			350:
				(*1.发送给上位机的数据*)
			//	WorkStation_TCP.PLC_SEND1.m_nMoveState	:=2;			//send[9]//0-准备过程中 1-准备完成 2-曝光中 3-本次扫描结束	
				(*1.给上位机发送的数*)
				IF Entity_IO.bXrayExp THEN
					WorkStation_TCP.PLC_SEND1.m_nExpStates	:=2;//
				END_IF;
				WorkStation_TCP.PLC_SEND1.m_nScanProType:=2;			//send[16]
				
				(*2.曝光结束，跳出*)
				IF DT_Xray.RadExp_Step=66 THEN
					Step_Air:=360;	
				END_IF
			
			360:
				(*1.运动变量复位*)
				Entity_IO.bXaryOne:=FALSE;
				Entity_IO.bXaryTwo:=FALSE;
				Axis_QJ.QJ_AxisCmd.bAbs:=FALSE;
				Axis_XZ.XZ_AxisCmd.bAbs:=FALSE;	
				Entity_IO.bTriggerOut:=FALSE;
	
				(*2.给上位机发送数据，不能太快*)
				TON_Air[36](IN:=TRUE , PT:=T#1600MS , Q=> , ET=> );	//留些时间给上位机发送本次扫描结束方案标志
				
				(*2.扫描结束，发送结束标志位*)
				IF DT_Xray.RadExp_Step=77 THEN 
					WorkStation_TCP.PLC_SEND1.m_nMoveState:=3;			//send[9] //0-准备过程中 1-准备完成 2-曝光中 3-本次扫描结束
				END_IF;
				
				(*3.判断师傅最后一次扫描*)
				IF TON_Air[36].Q THEN
					IF (WorkStation_TCP.PLC_RECV1.m_nCircleIndex+1)>=(WorkStation_TCP.PLC_RECV1.m_nCircleCount) AND bAirLast3 AND DT_Xray.RadExp_Step=77 THEN 	//用于区分自动扫是否最后一次，此时=1，=1都等于1
						GVL_SCAN.bJumpScan:=TRUE;
					END_IF;
				END_IF
				
				(*4.不是最后一次，收到下一次命令，继续扫*)
				IF WorkStation_TCP.PLC_RECV1.m_nSocketType=1 AND DT_Xray.RadExp_Step=77 THEN 	//增加第二次运动判断，m_nSocketType=1 
					Step_Air:=300;
				END_IF
	END_CASE
END_ACTION

TRANSITION T_AirCal:
(*进入空气校正/高清校正模式*)
	WorkStation_TCP.PLC_RECV1.m_nSocketType=1 AND (WorkStation_TCP.PLC_RECV1.m_nExpId=7  OR WorkStation_TCP.PLC_RECV1.m_nExpId=8)
END_TRANSITION

TRANSITION T_AirCal_Quick:
(*进入空气校正/快速校正模式*)
	WorkStation_TCP.PLC_RECV1.m_nSocketType=1 AND WorkStation_TCP.PLC_RECV1.m_nExpId=8
END_TRANSITION

ACTION _AirCalQuick_active:

	CASE Step_Air_Quick OF 
		300://快速扫描校正
				//初始化准备流程
				(*1.给上位机发送的数据*)
				WorkStation_TCP.PLC_SEND1.m_nMoveState:=0;			//send[9] //0-准备过程中 1-准备完成 2-曝光中 3-本次扫描结束 
				bAirLast3		:=FALSE;
				Entity_IO.bXraySwitch:=FALSE;//
				(*2.中间变量复位*)
				FOR i:=1 TO 50 BY 1 DO 
					TON_Air[i](IN:= FALSE);
				END_FOR
				Axis_XZ.XZ_AxisCmd.bAbs		:=FALSE;
				Axis_QJ.QJ_AxisCmd.bAbs		:=FALSE;
				Step_Air_Quick:=310;
				
			310:
				(*1.发送给上位机的数据*)
				WorkStation_TCP.PLC_SEND1.m_nExpStates	:=1;		//0-准备过程中 1-准备完成 2-曝光中 3-本次扫描结束	
				WorkStation_TCP.PLC_SEND1.m_nMoveState	:=0;		//起始、终止状态， 默认值0， 1为当前扫描方案处于准备好状态，可以准备扫描；2为当前扫描方案结束，运动过程中值为0
				WorkStation_TCP.PLC_SEND1.m_nScanProType:=2;		//扫描方案类型 , 1-手动，0-自动. 
			
				(*2.旋转轴和前进轴自动运动到目标位置*)
				(*2.1 旋转轴直接运动到目标位置*)
				Axis_XZ.XZ_AxisCmd.AxisPara.rAbsPosition	:=LIMIT(-3,WorkStation_TCP.PLC_RECV1.m_nRotateBegin,363);
				Axis_XZ.XZ_AxisCmd.AxisPara.rAbsVelocity	:=30;
				TON_Air[31](IN:=TRUE , PT:=T#500MS);
				Axis_XZ.XZ_AxisCmd.bAbs						:=TON_Air[31].Q;
	
				(*2.2 前进轴直接运动到目标位置*)
				Axis_QJ.QJ_AxisCmd.AxisPara.rAbsPosition	:=LIMIT(0,WorkStation_TCP.PLC_RECV1.m_fScanTop,900);
				Axis_QJ.QJ_AxisCmd.AxisPara.rAbsVelocity	:=60;
				TON_Air[32](IN:=TRUE , PT:=T#500MS);
				Axis_QJ.QJ_AxisCmd.bAbs						:=TON_Air[32].Q;
				
				(*5.跳转*)
				TON_Air[33](IN:=ABS(Axis_QJ.QJ_AxisState.rActPosition-WorkStation_TCP.PLC_RECV1.m_fScanTop)<1 
					AND ABS(Axis_XZ.XZ_AxisState.rActPosition-WorkStation_TCP.PLC_RECV1.m_nRotateBegin)<1 
					AND Axis_XZ.XZ_AxisState.bStandStill AND Axis_QJ.QJ_AxisState.bStandStill, PT:=T#150MS);
				IF TON_Air[33].Q THEN  
					Step_Air_Quick:=320;
				END_IF
				
			320://写入射线源参数成功
				(*1.变量复位*)
				Axis_XZ.XZ_AxisCmd.bAbs		:=FALSE;
				Axis_QJ.QJ_AxisCmd.bAbs		:=FALSE;
				
				(*2.射线源参数写入正常完毕*)
				IF DT_Xray.ExpPara_Step=66 THEN
					Step_Air_Quick:=330;
				END_IF
				
			330:
				//扫描中间态，跳转使用
				(*1.变量复位*)
				FOR i:=1 TO 50 BY 1 DO 
					TON_Air[i](IN:= FALSE);
				END_FOR
				Axis_QJ.QJ_AxisCmd.bAbs:=FALSE;//复位前进轴
				Axis_XZ.XZ_AxisCmd.bAbs:=FALSE;//复位旋转轴
				Step_Air_Quick:=340;
				
			340://开启曝光
				(*1.发送给上位机的数据*)
				WorkStation_TCP.PLC_SEND1.m_nMoveState	:=1;	//send[9]
				WorkStation_TCP.PLC_SEND1.m_nScanProType:=2;	//send[16]
				
				(*2.射线源参数写入成功，开启透视*)
				IF DT_Xray.ExpPara_Step=66 THEN  //保证写入参数
					Entity_IO.bXaryOne:=TRUE;//开启一二档
					Entity_IO.bXaryTwo:=TRUE;//开启一二档
				END_IF;
				
				(*3.判断是否最后一次扫描*)
				IF WorkStation_TCP.PLC_RECV1.m_nLastMsg=1 THEN
					bAirLast3 := TRUE;
				ELSE
					bAirLast3 := FALSE;
				END_IF
				
				(*4.跳转指令*)
				TON_Air[34](IN:=TRUE,PT:=T#2600MS);//把曝光的时间加这这里了
				IF TON_Air[34].Q AND Entity_IO.bXaryOne AND Entity_IO.bXaryTwo THEN
					Step_Air_Quick:=350;
				END_IF
				
			350:
				(*1.发送给上位机的数据*)
				WorkStation_TCP.PLC_SEND1.m_nMoveState	:=2;			//send[9]//0-准备过程中 1-准备完成 2-曝光中 3-本次扫描结束	
				WorkStation_TCP.PLC_SEND1.m_nScanProType:=2;			//send[16]
				
				(*2.曝光结束，跳出*)
				IF DT_Xray.RadExp_Step=66 THEN
					Step_Air_Quick:=360;	
				END_IF
			
			360:
				(*1.运动变量复位*)
				Entity_IO.bXaryOne:=FALSE;
				Entity_IO.bXaryTwo:=FALSE;
				Axis_QJ.QJ_AxisCmd.bAbs:=FALSE;
				Axis_XZ.XZ_AxisCmd.bAbs:=FALSE;	
				Entity_IO.bTriggerOut:=FALSE;
	
				(*2.给上位机发送数据，不能太快*)
				TON_Air[36](IN:=TRUE , PT:=T#1600MS , Q=> , ET=> );	//留些时间给上位机发送本次扫描结束方案标志
				
				(*2.扫描结束，发送结束标志位*)
				IF DT_Xray.RadExp_Step=77 THEN 
					WorkStation_TCP.PLC_SEND1.m_nMoveState:=3;			//send[9] //0-准备过程中 1-准备完成 2-曝光中 3-本次扫描结束
				END_IF;
				
				(*3.判断师傅最后一次扫描*)
				IF TON_Air[36].Q THEN
					IF (WorkStation_TCP.PLC_RECV1.m_nCircleIndex+1)>=(WorkStation_TCP.PLC_RECV1.m_nCircleCount) AND bAirLast3 AND DT_Xray.RadExp_Step=77 THEN 	//用于区分自动扫是否最后一次，此时=1，=1都等于1
						GVL_SCAN.bJumpScan:=TRUE;
					END_IF;
				END_IF
				
				(*4.不是最后一次，收到下一次命令，继续扫*)
				IF WorkStation_TCP.PLC_RECV1.m_nSocketType=1 AND DT_Xray.RadExp_Step=77 THEN 	//增加第二次运动判断，m_nSocketType=1 
					Step_Air_Quick:=300;
				END_IF
		END_CASE
END_ACTION

ACTION _AirCalQuick_entry:
Step_Air_Quick:=300; 

GVL_State.iPLC_State:=350;//空气校正
END_ACTION

ACTION _AirCalHign_exit:


	Entity_IO.bTriggerOut:=FALSE;
	Entity_io.bXraySwitch:=FALSE;//PF CLK信号切换继电器 不得电是默认BUCKY触发
	
	iTriggerNum1:=0;
	iTriggerNum2:=0;
END_ACTION

ACTION _AirCalQuick_exit:

END_ACTION

ACTION _a_Debug_exit:


Entity_IO.bXaryFlu:=FALSE;
END_ACTION

ACTION _a_Emergercy_exit:

Axis_XZ.XZ_AxisCmd.bReset:=TRUE;
Axis_QJ.QJ_AxisCmd.bReset:=TRUE;
END_ACTION

ACTION _ModeWait_active:

IF Axis_XZ.XZ_AxisCmd.bPower=FALSE THEN 
	Axis_XZ.XZ_AxisCmd.bPower:=TRUE;
ELSE
	;
END_IF

IF Axis_QJ.QJ_AxisCmd.bPower=FALSE THEN 
	Axis_QJ.QJ_AxisCmd.bPower:=TRUE;
ELSE
	;
END_IF
END_ACTION

END_PROGRAM

// Device/Application/Refer/XRAY_RS485
PROGRAM XRAY_RS485
VAR
	Open_0: COM.Open;Hulala:BOOL;
	Write_0: COM.Write;
	Read_0: COM.Read;
	Close_0: COM.Close;
	xOpen_Exe:BOOL;
	hComHandle:CAA.HANDLE;
	byWrite2:ARRAY [0..3] OF BYTE;
	byWrite3:ARRAY [0..4] OF BYTE;
	byWrite4:ARRAY [0..5] OF BYTE;
	byWrite5:ARRAY [0..6] OF BYTE;
	byWrite6:ARRAY [0..7] OF BYTE;
	byWrite7:ARRAY [0..8] OF BYTE;
	byWrite8:ARRAY [0..9] OF BYTE;
	byWrite9:ARRAY [0..10] OF BYTE;
	xWrite_Exe:BOOL;
	xRead_Exe:BOOL;
    byReadData:ARRAY [0..255] OF BYTE;
    xClose_Exe:BOOL;
	aParamsB19200 : ARRAY [1..7] OF COM.PARAMETER := [
    (udiParameterId := COM.CAA_Parameter_Constants.udiPort,udiValue := 3), 					//指令端口2,3,4,5分别对应硬件接口com2、com0、com1、com3
    (udiParameterId := COM.CAA_Parameter_Constants.udiBaudrate,udiValue := 19200),			//波特率，设置为19200
    (udiParameterId := COM.CAA_Parameter_Constants.udiParity,udiValue := COM.PARITY.NONE),	//校验，设置为无校验
    (udiParameterId := COM.CAA_Parameter_Constants.udiStopBits,udiValue := COM.STOPBIT.ONESTOPBIT),//停止位，1位
    (udiParameterId := COM.CAA_Parameter_Constants.udiTimeout,udiValue := 500),				//超时时间，设置成500ms
    (udiParameterId := COM.CAA_Parameter_Constants.udiByteSize,udiValue := 8),				//数据位
    (udiParameterId := COM.CAA_Parameter_Constants.udiBinary, udiValue := 1)				//二进制参数，启用二进制模式
];		
	TON1,TON2:Standard.TON;
	bSend:BOOL;
	iSize	:INT;
	String2Byte1:String2Byte;
	sSendString:STRING;//
	BLINK1,BLINK2:Blink;
//	Main_Step,Init_Step,DefaultPara_Step,Standby_Step,Rad_Step,Lookup_Step:UINT;
	sRecvString:ARRAY [0..9] OF STRING;	
	sRecvByte:ARRAY [0..39] OF BYTE;	
	i:INT;
	RecvNum,RecvNum1:INT;
	ASCII_Chart_N1:ARRAY [0..9] OF ASCII_Chart_N;
	sRecvStringA1,sRecvStringA2,sRecvStringA3,sRecvStringA4:STRING;
	sRecvStringA5,sRecvStringA6,sRecvStringA7,sRecvStringA0:STRING;
	R_TRIG1:Standard.R_TRIG;
	R30_0,R30_1,R30_2,R30_3,R30_4,R30_5,R30_6:Standard.R_TRIG;
	R10,R20,R30,R40,R50,R60:Standard.R_TRIG;
	TON0_20,TON30_0,TON30_20,TON30_30:Standard.TON;
	f10:F_TRIG;
	BLINK1_ST,BLINK11: BLINK;
	TEMP_MA:UINT;
	TEMP_MS: UINT;
	TON3,TON_ST,TON40,TON_FLR:TON;
	ASCII_Chart_N2:ARRAY[0..30] OF ASCII_Chart_N;
	ASCII_Chart_N_Alarm:ARRAY[0..5] OF ASCII_Chart_N;
	TEMP_FLX1:BOOL;
	TON22:TON;
	R_JUMP20:R_TRIG;
	TON33: TON;
	TON_DelayPara:TON;
	HULALA111:BOOL;
	
	TON11,TON12:TON;
	TON_KV,TON_MA:Standard.TON; //参数设置不对后，延迟进行报警处理0228
	Booting: BOOL;
	hlaldjlk: BOOL;
	Feedback_mA1:REAL;
	Feedback_Kv1:UDINT;
	TON_DELAY:TON;
	
	XXX:X_RayFluPara;
	aaa1:ARRAY[1..255] OF BYTE;
	aaa:ARRAY[1..255] OF BYTE;
	
ddd:UINT;
Error:INT;
j:INT;
xxxxx:String_TO_ASCII;
	CheckSum:UINT;
	CheckSum1: UINT;
	CheckSum3:STRING;
	sSendStringX:STRING;
	
	
	ReadString:RecvStringS;
	
	
END_VAR

VAR_INPUT
	
END_VAR

VAR_OUTPUT
	Main_Step,Init_Step,DefaultPara_Step,Standby_Step,Rad_Step,Lookup_Step:UINT;
	Feedback_Kv:UDINT;
	Feedback_mA:REAL;
	Feedback_ms:REAL;
	Feedback_nFocus:UDINT;
	Feedback_nMHuValue:REAL;
	Feedback_AccTime:REAL;
	iAlarmNum:UINT;		//射线源部分的报警位
END_VAR

(*README*)
(*射线源通讯子功能块*)

(*---------------------------------------------------第一部分：串口参数设置------------------------------------------------*)
(*1.open*)
	TON1(IN:=TRUE , PT:=T#5S);//开机后5秒打开串口
	Open_0(xExecute:=TON1.Q , xDone=> , xBusy=> , xError=> , usiListLength:=20 , pParameterList:=ADR(aParamsB19200) , eError=> , hCom=>hComHandle );

	
(*2.Write*)
	Write_0(
			xExecute:= Open_0.xDone AND bSend, 
			xAbort:= , 
			udiTimeOut:=500 , 
			xDone=> , 
			xBusy=> , 
			xError=> , 
			xAborted=> , 
			hCom:= hComHandle, 
			pBuffer:= , //后面写的
			szSize:= , 
			eError=> );	
			
(*3.Read*)
	TON2(IN:=NOT TON2.Q , PT:=T#20MS , Q=> , ET=> );	//射线源周期100ms
	Read_0(
			xExecute:= Open_0.xDone AND TON2.Q AND NOT(bSend),
			xAbort:= , 
			udiTimeOut:= 500, 
			xDone=> , 
			xBusy=> , 
			xError=> , 
			xAborted=> , 
			hCom:= hComHandle, 
			pBuffer:= ADR(byReadData), 
			szBuffer:= 10, 
			eError=> , 
			szSize=> );
	
(*4.Close*)
	Close_0(
			xExecute:= xClose_Exe, 
			xDone=> , 
			xBusy=> , 
			xError=> , 
			hCom:= hComHandle, 
			eError=> );

(*--------------------------------------------第二部分，数据处理--------------------------------------------------*)
(*2.1 写入命令处理*)
	iSize:=LIMIT(0,LEN(sSendString),255); 		//获取写入的字符串长度	已增加03H结束符+CheckSum和校验	
	Write_0.szSize:=INT_TO_USINT(iSize);
	Write_0.pBuffer:=ADR(sSendString);

	XXX( 
	WS:= 1, 
	FLF:= 2, 
	FLA:=0 , 
	FLS:=195 , 
	FLR:=1 , 
	FLK:= 090, 
	FLM:= 060, 
	Out=> );
	
	sSendStringX:=XXX.Out;

xxxxx(
		InputString:=XXX.Out , 
		MaxArraySize:= 255, 
		ASCIIArray=> aaa1, 
		ArrayLength=> , 
		Error=> , 
		ErrorMessage=> );
		
	CheckSum:=0;
	FOR j:=1 TO 255 BY 1 DO
		IF aaa1[j]=16#20 THEN   	//空格对应的ASCII码不计入和校验中
			CONTINUE;
		END_IF
		CheckSum:=CheckSum+aaa1[j];
	END_FOR

	CheckSum1:=(CheckSum) AND 16#FF; 	//取低字节byte
	IF CheckSum1<16 THEN 
		NumToHexString(In:= CheckSum1, L:=1, Fill:=LS_OmronUtils._eFILL_CHR._ZERO, Out=> CheckSum3);
	ELSE
		NumToHexString(In:= CheckSum1, L:=2, Fill:=LS_OmronUtils._eFILL_CHR._NULL, Out=> CheckSum3);
	END_IF
	
	sSendString:=CONCAT(STR1:=sSendStringX , STR2:= CheckSum3);


	ReadString(Excute:= Read_0.xDone AND Read_0.szSize<>0, Size:=__UXINT_TO_INT(Read_0.szSize) , RecvArray:=byReadData , RecvString=>sRecvStringA0 );









(*

(*2.1 写入命令处理*)
	iSize:=LIMIT(0,LEN(sSendString),10); 		//获取写入的字符串长度	已增加03H结束符+CheckSum和校验	
	String2Byte1(sXrayString:=sSendString , sByte=> );
	Write_0.szSize:=INT_TO_USINT(iSize)+2;
	CASE iSize OF 
	2:
		(*2个字符的命令*)	
		byWrite2[0]:=String2Byte1.sByte[1];
		byWrite2[1]:=String2Byte1.sByte[2];
		byWrite2[2]:=16#03;
		byWrite2[3]:=byWrite2[0]+byWrite2[1]+byWrite2[2];
		Write_0.pBuffer:=ADR(byWrite2);
	3:	
		(*3个字符的命令*)	
		byWrite3[0]:=String2Byte1.sByte[1];
		byWrite3[1]:=String2Byte1.sByte[2];
		byWrite3[2]:=String2Byte1.sByte[3];
		byWrite3[3]:=16#03;
		byWrite3[4]:=byWrite3[0]+byWrite3[1]+byWrite3[2]+byWrite3[3];
		Write_0.pBuffer:=ADR(byWrite3);
	
	4:
		(*4个字符的命令*)	
		byWrite4[0]:=String2Byte1.sByte[1];
		byWrite4[1]:=String2Byte1.sByte[2];
		byWrite4[2]:=String2Byte1.sByte[3];
		byWrite4[3]:=String2Byte1.sByte[4];
		byWrite4[4]:=16#03;
		byWrite4[5]:=byWrite4[0]+byWrite4[1]+byWrite4[2]+byWrite4[3]+byWrite4[4];
		Write_0.pBuffer:=ADR(byWrite4);
	
	5:
		(*5个字符的命令*)	
		byWrite5[0]:=String2Byte1.sByte[1];
		byWrite5[1]:=String2Byte1.sByte[2];
		byWrite5[2]:=String2Byte1.sByte[3];
		byWrite5[3]:=String2Byte1.sByte[4];
		byWrite5[4]:=String2Byte1.sByte[5];
		byWrite5[5]:=16#03;
		byWrite5[6]:=byWrite5[0]+byWrite5[1]+byWrite5[2]+byWrite5[3]+byWrite5[4]+byWrite5[5];
		Write_0.pBuffer:=ADR(byWrite5);
		
	6:
		(*6个字符的命令*)	
		byWrite6[0]:=String2Byte1.sByte[1];
		byWrite6[1]:=String2Byte1.sByte[2];
		byWrite6[2]:=String2Byte1.sByte[3];
		byWrite6[3]:=String2Byte1.sByte[4];
		byWrite6[4]:=String2Byte1.sByte[5];
		byWrite6[5]:=String2Byte1.sByte[6];
		byWrite6[6]:=16#03;
		byWrite6[7]:=byWrite6[0]+byWrite6[1]+byWrite6[2]+byWrite6[3]+byWrite6[4]+byWrite6[5]+byWrite6[6];
		Write_0.pBuffer:=ADR(byWrite6);		
	7:
		(*7个字符的命令*)	
		byWrite7[0]:=String2Byte1.sByte[1];
		byWrite7[1]:=String2Byte1.sByte[2];
		byWrite7[2]:=String2Byte1.sByte[3];
		byWrite7[3]:=String2Byte1.sByte[4];
		byWrite7[4]:=String2Byte1.sByte[5];
		byWrite7[5]:=String2Byte1.sByte[6];
		byWrite7[6]:=String2Byte1.sByte[7];
		byWrite7[7]:=16#03;
		byWrite7[8]:=byWrite7[0]+byWrite7[1]+byWrite7[2]+byWrite7[3]+byWrite7[4]+byWrite7[5]+byWrite7[6]+byWrite7[7];
		Write_0.pBuffer:=ADR(byWrite7);
		
	8:(*8个字符的命令*)	
		byWrite8[0]:=String2Byte1.sByte[1];
		byWrite8[1]:=String2Byte1.sByte[2];
		byWrite8[2]:=String2Byte1.sByte[3];
		byWrite8[3]:=String2Byte1.sByte[4];
		byWrite8[4]:=String2Byte1.sByte[5];
		byWrite8[5]:=String2Byte1.sByte[6];
		byWrite8[6]:=String2Byte1.sByte[7];
		byWrite8[7]:=String2Byte1.sByte[8];
		byWrite8[8]:=16#03;
		byWrite8[9]:=byWrite8[0]+byWrite8[1]+byWrite8[2]+byWrite8[3]+byWrite8[4]+byWrite8[5]+byWrite8[6]+byWrite8[7]+byWrite8[8];
		Write_0.pBuffer:=ADR(byWrite8);
	ELSE
		;//输入错误
	END_CASE
	
*)		
	(*2.2 读取命令*)
(*	sRecvByte:=byReadData;

	R_TRIG1(CLK:=Read_0.xDone AND Read_0.szSize<>0, Q=> );		//获取读到了多少个字符
	IF R_TRIG1.Q THEN
		RecvNum:=LIMIT(0,__UXINT_TO_INT(Read_0.szSize)-2,9);	//限制了一下字符0124
	END_IF;

	FOR i:=0 TO RecvNum BY 1 DO 
		ASCII_Chart_N1[i](byASCII:=sRecvByte[i] , sOut_Single=>sRecvString[i] );//需要调用功能块才能有输出
	END_FOR 

	CASE RecvNum OF 		//最长8个字符,如遇到RS和RR的反馈，就自己数字节吧，这里给反馈命令使用
		0:
			sRecvStringA0:='NULL';
		1:
			sRecvStringA0:=sRecvString[0];
		2:
			sRecvStringA0:=CONCAT(STR1:=sRecvString[0] , STR2:= sRecvString[1]);
		3:
			sRecvStringA1:=CONCAT(STR1:=sRecvString[0] , STR2:= sRecvString[1]);
			sRecvStringA0:=CONCAT(STR1:=sRecvStringA1 , STR2:= sRecvString[2]);
		4:
			sRecvStringA1:=CONCAT(STR1:=sRecvString[0] , STR2:= sRecvString[1]);
			sRecvStringA2:=CONCAT(STR1:=sRecvString[2] , STR2:= sRecvString[3]);
			sRecvStringA0:=CONCAT(STR1:=sRecvStringA1 , STR2:= sRecvStringA2);
		5:
			sRecvStringA1:=CONCAT(STR1:=sRecvString[0] , STR2:= sRecvString[1]);
			sRecvStringA2:=CONCAT(STR1:=sRecvString[2] , STR2:= sRecvString[3]);
			sRecvStringA3:=CONCAT(STR1:=sRecvStringA1 , STR2:= sRecvStringA2);
			sRecvStringA0:=CONCAT(STR1:=sRecvStringA3 , STR2:= sRecvString[4]);
		6:
			sRecvStringA1:=CONCAT(STR1:=sRecvString[0] , STR2:= sRecvString[1]);
			sRecvStringA2:=CONCAT(STR1:=sRecvString[2] , STR2:= sRecvString[3]);
			sRecvStringA3:=CONCAT(STR1:=sRecvString[4] , STR2:= sRecvString[5]);
			sRecvStringA4:=CONCAT(STR1:=sRecvStringA1 , STR2:= sRecvStringA2);
			sRecvStringA0:=CONCAT(STR1:=sRecvStringA4 , STR2:= sRecvStringA3);
		7:
			sRecvStringA1:=CONCAT(STR1:=sRecvString[0] , STR2:= sRecvString[1]);
			sRecvStringA2:=CONCAT(STR1:=sRecvString[2] , STR2:= sRecvString[3]);
			sRecvStringA3:=CONCAT(STR1:=sRecvString[4] , STR2:= sRecvString[5]);
			sRecvStringA4:=CONCAT(STR1:=sRecvStringA1 , STR2:= sRecvStringA2);
			sRecvStringA5:=CONCAT(STR1:=sRecvStringA4 , STR2:= sRecvStringA3);
			sRecvStringA0:=CONCAT(STR1:=sRecvStringA5 , STR2:= sRecvString[6]);
		8:
			sRecvStringA1:=CONCAT(STR1:=sRecvString[0] , STR2:= sRecvString[1]);
			sRecvStringA2:=CONCAT(STR1:=sRecvString[2] , STR2:= sRecvString[3]);
			sRecvStringA3:=CONCAT(STR1:=sRecvString[4] , STR2:= sRecvString[5]);
			sRecvStringA4:=CONCAT(STR1:=sRecvString[6] , STR2:= sRecvString[7]);
			sRecvStringA5:=CONCAT(STR1:=sRecvStringA1 , STR2:= sRecvStringA2);
			sRecvStringA6:=CONCAT(STR1:=sRecvStringA3 , STR2:= sRecvStringA4);
			sRecvStringA0:=CONCAT(STR1:=sRecvStringA5 , STR2:= sRecvStringA6);
		9:
			sRecvStringA1:=CONCAT(STR1:=sRecvString[0] , STR2:= sRecvString[1]);
			sRecvStringA2:=CONCAT(STR1:=sRecvString[2] , STR2:= sRecvString[3]);
			sRecvStringA3:=CONCAT(STR1:=sRecvString[4] , STR2:= sRecvString[5]);
			sRecvStringA4:=CONCAT(STR1:=sRecvString[6] , STR2:= sRecvString[7]);
			sRecvStringA5:=CONCAT(STR1:=sRecvStringA1 , STR2:= sRecvStringA2);
			sRecvStringA6:=CONCAT(STR1:=sRecvStringA3 , STR2:= sRecvStringA4);
			sRecvStringA7:=CONCAT(STR1:=sRecvStringA5 , STR2:= sRecvStringA6);
			sRecvStringA0:=CONCAT(STR1:=sRecvStringA7 , STR2:= sRecvString[8]);
		ELSE
			sRecvStringA0:='Too Long';
	END_CASE
*)
(*3.射线源状态机处理*)	
//	AXray( );
//	GVL_State.iXray_State:=UINT_TO_BYTE(Main_Step);//获取射线源状态

ACTION AXray:

(*---------------------------------------------第三部分：射线源状态机---------------------------------------------------*)
(*0.公共部分*)
(*	BLINK1(ENABLE:=TON1.Q , TIMELOW:=T#300MS , TIMEHIGH:=T#200MS , OUT=> );
	BLINK1_ST(ENABLE:=TON1.Q , TIMELOW:=T#2S , TIMEHIGH:=T#2S , OUT=> );
	
	(*1.初始化阶段，Initialization Phase*)
			CASE Main_Step OF 
				0:	(*1.初始化阶段，Initialization Phase*)
				IF (sRecvByte[0]= 16#45 AND sRecvByte[1]= 16#4C) OR sRecvStringA0='ST008' THEN //收到ER或EL,确认收到了错误信号，ER可以理解为可恢复，EL为不可恢复 收到EL信号可复位，ER信号只是显示
						Main_Step:=40;
				ELSE
					CASE Init_Step OF 
					0:	//参数初始化
						bSend			:=FALSE;
						DefaultPara_Step:=0;
						Standby_Step	:=0;
						Rad_Step		:=0;//射线步骤复位
						TON11(IN:= TRUE, PT:=T#3S);//开机延迟
						IF TON11.Q THEN
							Init_Step		:=10;
						END_IF
						
					10:	//建立通讯
						TON11(IN:= FALSE);
						sSendString:='ST';
						bSend:=BLINK1_ST.OUT;  
						IF sRecvStringA0='ST001' OR sRecvStringA0='ST002' THEN //收到ST000，通讯正常//此版本是001，所有状态都加1，文档状态说明都加1
							Init_Step:=20;
						ELSE
							iAlarmNum:=301;		//通讯错误
						END_IF
						
					20://检查错误,如果有错误，就复位，没错误，延迟2秒跳转
						iAlarmNum:=0;		//通讯
						IF sRecvByte[0]= 16#45 AND (sRecvByte[1]= 16#4C) THEN //收到ER或EL,确认收到了错误信号，EL可以理解为可恢复，ER为不可恢复 收到EL信号可复位，ER信号只是显示
							sSendString:=sRecvStringA0;
							bSend:=BLINK1.OUT;
							TON0_20(IN:=FALSE);
						ELSE
							TON0_20(IN:=TRUE , PT:=T#2S);//2秒内无报错
							IF TON0_20.Q THEN
								sSendString:='ST';
								bSend:=BLINK1.OUT;
								IF sRecvStringA0='ST002' OR sRecvStringA0='ST001' THEN //收到ST002，通讯正常//此版本是001，所有状态都加1
									Init_Step:=66;
								END_IF
							END_IF;
						END_IF
					66:
						Main_Step:=10;
					ELSE
						;
					END_CASE
				END_IF;
				
				10:	(*写入默认参数，开机只写一次*)	
					IF (sRecvByte[0]= 16#45 AND sRecvByte[1]= 16#4C) OR sRecvStringA0='ST008' THEN //收到ER或EL,确认收到了错误信号，ER可以理解为可恢复，EL为不可恢复 收到EL信号可复位，ER信号只是显示
						Main_Step:=40;
					ELSE
						CASE DefaultPara_Step OF 
						0:
							bSend:=FALSE;
							TON_DelayPara(IN:=FALSE);
							DefaultPara_Step:=5;
					
						5:
							TON_DelayPara(IN:=TRUE , PT:=T#5S , Q=> , ET=> );//写默认参数的时候需要等等射线源一些时间
							IF TON_DelayPara.Q THEN
								DefaultPara_Step:=10;
							END_IF
							
						10://1.关闭AEC
							TON_DelayPara(IN:=FALSE);
							sSendString:='FI000';
							bSend:=BLINK1.OUT;
							IF sRecvStringA0='FI000' THEN
								DefaultPara_Step:=20;
							END_IF
							
						20:
							sSendString:='ET1';
							bSend:=BLINK1.OUT;
							IF sRecvStringA0='ET1' THEN
								DefaultPara_Step:=30;
							END_IF
							
						30://工作模式选择
							sSendString:='WS1';
							bSend:=BLINK1.OUT;
							IF sRecvStringA0='WS1' THEN
								DefaultPara_Step:=40;
							END_IF
						40:
							bSend:=FALSE;
							Main_Step:=20;
						ELSE 
							;
						END_CASE
					END_IF;
		
				20:	(*静止等待状态，Standby Phase*)//注意增加ST，每5秒的周期
					Rad_Step	:=0;
					IF (sRecvByte[0]= 16#45 AND sRecvByte[1]= 16#4C) OR sRecvStringA0='ST008' THEN //收到ER或EL,确认收到了错误信号，ER可以理解为可恢复，EL为不可恢复 收到EL信号可复位，ER信号只是显示
						Main_Step:=40;	
					ELSE
						iAlarmNum:=0;//复位故障	
						IF GVL_State.iPLC_State=40 AND GVL_State.bBooting THEN
							Standby_Step:=10;
						ELSE
							CASE Standby_Step OF
								0:
									bSend		:=FALSE;
									Rad_Step	:=0;//射线步骤复位
									Standby_Step:=9;
									TON33(IN:= FALSE);
									
								9:
									IF sRecvStringA0='FLP0' THEN
										sSendString:='FLP0';
									ELSE
										;
									END_IF	
									R30_0(CLK:=(sRecvStringA0='FLP0') AND Read_0.xDone, Q=> );
									bSend:=R30_0.Q;
		
									TON33(IN:= TRUE, PT:= T#300MS, Q=> , ET=> );
									IF TON33.Q THEN
										Standby_Step:=10;
									END_IF
									
								10://查询指令
									TON33(IN:= FALSE);
									IF (WorkStation_TCP.PLC_RECV1.m_nSocketType=0)  		//=0的时候不写参数
										OR (WorkStation_TCP.PLC_RECV1.m_nControlState>=1 AND WorkStation_TCP.PLC_RECV1.m_nSocketType=1)	//强制退出的时候不写参数
										OR (WorkStation_TCP.PLC_RECV1.m_nExpId=5 		 AND WorkStation_TCP.PLC_RECV1.m_nSocketType=1)	//状态=5的时候不写参数 250701
											 THEN  //开启查询，5秒不能断//可以在这里增加空气校正的条件，例如 OR GVL_State.iPLC_State=控制校正
										CASE Lookup_Step OF 
											0:
												sSendString:='ST';//
												IF BLINK1_ST.OUT THEN
													Lookup_Step:=1;
												END_IF
											1:
												sSendString:='FLK?';//当前电压
												IF BLINK1_ST.OUT THEN
													Lookup_Step:=2;
												END_IF
											2:
												sSendString:='FLM?';//当前电流
												IF BLINK1_ST.OUT THEN
													Lookup_Step:=3;
												END_IF
											3:
												sSendString:='FLT?';//当前透视累计时间
												IF BLINK1_ST.OUT THEN
													Lookup_Step:=4;
												END_IF
											4:
												sSendString:='HE?';//当前球管热量HE
												IF BLINK1_ST.OUT THEN
													Lookup_Step:=5;
												END_IF
											5:
												sSendString:='RF';//透视下的信息
												IF BLINK1_ST.OUT THEN
													Lookup_Step:=0;
												END_IF
										END_CASE
										bSend:=BLINK1_ST.OUT;	//2秒查询一次	
										(*数据解析*)
										IF sRecvByte[0]=16#46 AND sRecvByte[1]=16#4C AND sRecvByte[2]=16#4B THEN //FLK 电压
											ASCII_Chart_N2[0](byASCII:= sRecvByte[3], sOut_Single=> );
											ASCII_Chart_N2[1](byASCII:= sRecvByte[4], sOut_Single=> );
											ASCII_Chart_N2[2](byASCII:= sRecvByte[5], sOut_Single=> );
											Feedback_Kv1:=STRING_TO_UDINT(ASCII_Chart_N2[0].sOut_Single)*100+STRING_TO_UDINT(ASCII_Chart_N2[1].sOut_Single)*10+STRING_TO_UDINT(ASCII_Chart_N2[2].sOut_Single);
										END_IF
										
										IF sRecvByte[0]=16#46 AND sRecvByte[1]=16#4C AND sRecvByte[2]=16#4D THEN //FLM 电流
											ASCII_Chart_N2[0](byASCII:= sRecvByte[3], sOut_Single=> );
											ASCII_Chart_N2[1](byASCII:= sRecvByte[4], sOut_Single=> );
											ASCII_Chart_N2[2](byASCII:= sRecvByte[5], sOut_Single=> );
											Feedback_mA1:=STRING_TO_REAL(ASCII_Chart_N2[0].sOut_Single)*10+STRING_TO_REAL(ASCII_Chart_N2[1].sOut_Single)*1+STRING_TO_REAL(ASCII_Chart_N2[2].sOut_Single)*0.1;
										END_IF 
										
										IF sRecvByte[0]=16#46 AND sRecvByte[1]=16#4C AND sRecvByte[2]=16#54 THEN //FLT 累计时间
											ASCII_Chart_N2[0](byASCII:= sRecvByte[3], sOut_Single=> );
											ASCII_Chart_N2[1](byASCII:= sRecvByte[4], sOut_Single=> );
											ASCII_Chart_N2[2](byASCII:= sRecvByte[5], sOut_Single=> );
											Feedback_AccTime:=STRING_TO_REAL(ASCII_Chart_N2[0].sOut_Single)*10+STRING_TO_REAL(ASCII_Chart_N2[1].sOut_Single)*1+STRING_TO_REAL(ASCII_Chart_N2[2].sOut_Single)*0.1;
										END_IF 
										
										IF sRecvByte[0]=16#48 AND sRecvByte[1]=16#45 THEN //HE 球管热量
											ASCII_Chart_N2[0](byASCII:= sRecvByte[2], sOut_Single=> );
											ASCII_Chart_N2[1](byASCII:= sRecvByte[3], sOut_Single=> );
											ASCII_Chart_N2[2](byASCII:= sRecvByte[4], sOut_Single=> );
											Feedback_nMHuValue:=STRING_TO_REAL(ASCII_Chart_N2[0].sOut_Single)*100+STRING_TO_REAL(ASCII_Chart_N2[1].sOut_Single)*10+STRING_TO_REAL(ASCII_Chart_N2[2].sOut_Single);
										END_IF
										TON_KV(IN:=FALSE);
										TON_MA(IN:=FALSE);
										
										IF sRecvByte[0]=16#46 AND sRecvByte[1]=16#4C AND sRecvByte[2]=16#4B THEN // RF的FLK电压反馈
											ASCII_Chart_N2[0](byASCII:= sRecvByte[3], sOut_Single=> );
											ASCII_Chart_N2[1](byASCII:= sRecvByte[4], sOut_Single=> );
											ASCII_Chart_N2[2](byASCII:= sRecvByte[5], sOut_Single=> );
											Feedback_Kv:=STRING_TO_UDINT(ASCII_Chart_N2[0].sOut_Single)*100+STRING_TO_UDINT(ASCII_Chart_N2[1].sOut_Single)*10+STRING_TO_UDINT(ASCII_Chart_N2[2].sOut_Single);
										END_IF
										
										IF sRecvByte[7]=16#46 AND sRecvByte[8]=16#4C AND sRecvByte[9]=16#4D THEN //RF的FLM电流反馈
											ASCII_Chart_N2[0](byASCII:= sRecvByte[10], sOut_Single=> );
											ASCII_Chart_N2[1](byASCII:= sRecvByte[11], sOut_Single=> );
											ASCII_Chart_N2[2](byASCII:= sRecvByte[12], sOut_Single=> );
											Feedback_mA:=STRING_TO_REAL(ASCII_Chart_N2[0].sOut_Single)*10+STRING_TO_REAL(ASCII_Chart_N2[1].sOut_Single)*1+STRING_TO_REAL(ASCII_Chart_N2[2].sOut_Single)*0.1;
										END_IF 
										 
									ELSE
										TON22(IN:= FALSE);
										Standby_Step:=24;
									END_IF
									
								20:	
									sSendString:='ET1';
									bSend:=BLINK1.OUT;
									IF sRecvStringA0='ET1' THEN
										Standby_Step:=21;
									END_IF
									
								21:
									sSendString:=CONCAT('FO',UDINT_TO_STRING(WorkStation_TCP.PLC_RECV1.m_nFocus));
									bSend:=BLINK1.OUT;
									IF sRecvStringA0=sSendString THEN
										Standby_Step:=22;
									END_IF
									
								22:
									sSendString:='EC9';
									bSend:=BLINK1.OUT;
									IF sRecvStringA0='EC9' THEN
										Standby_Step:=23;
									END_IF
									
								23:
									sSendString:='FLF0';
									bSend:=BLINK1.OUT;
									IF sRecvStringA0='FLF0' THEN
										Standby_Step:=24;
									END_IF
									
								24:
									TON_KV(IN:=FALSE);TON_MA(IN:=FALSE);
									sSendString:='FLS100';
									bSend:=BLINK1.OUT;
									IF sRecvStringA0='FLS100' THEN
										Standby_Step:=25;
									END_IF
									
								25:
									(*FLF2,脉冲透视模式，FLF1,连续脉冲模式，电流限制在0.5mA到6mA之间，80kV对应6mA,125KV对应4mA*)
									IF WorkStation_TCP.PLC_RECV1.m_nExpId=4 THEN	//新增脉冲连续模式0610
										sSendString:='FLF1';
									ELSE
										sSendString:='FLF2';
									END_IF
									bSend:=BLINK1.OUT;
									TON_FLR(IN:=FALSE);
									IF sRecvStringA0='FLF2' OR sRecvStringA0='FLF1' THEN
										Standby_Step:=28;
									END_IF
									
								28:	//清除累计时间指令
									sSendString:='FLR1';
									bSend:=BLINK1.OUT;
									TON_FLR(IN:=TRUE , PT:=T#1S , Q=> , ET=> );
									IF TON_FLR.Q OR sRecvStringA0='FLR' THEN
										Standby_Step:=40;
									END_IF
									
								40://写入管电压 小于100最高位补零
									IF WorkStation_TCP.PLC_RECV1.m_nKv>=100 THEN
										sSendString:=CONCAT('FLK',UDINT_TO_STRING(WorkStation_TCP.PLC_RECV1.m_nKv));
									ELSE
										sSendString:=CONCAT('FLK0',UDINT_TO_STRING(WorkStation_TCP.PLC_RECV1.m_nKv));
									END_IF
									bSend:=BLINK1.OUT;
									TEMP_MA:=0;
									
									IF sRecvStringA0=sSendString THEN
										Standby_Step:=50;
									END_IF	
									
									TON_KV(IN:=(sRecvStringA0<>sSendString) , PT:=T#5S , Q=> , ET=> );
									IF TON_KV.Q THEN
										WorkStation_TCP.PLC_SEND1.m_nExpStates	:=5;		//参数写入错误
									END_IF
									
									
								50://写入管电流 5位数字,0.1mA
									TEMP_MA:=LIMIT(1,REAL_TO_UINT(WorkStation_TCP.PLC_RECV1.m_nMA*10),10000);//获取发送过来的数，舍弃×10后的小数
									IF TEMP_MA>=10000 THEN
										sSendString:=CONCAT('FLM',UINT_TO_STRING(TEMP_MA));
									ELSIF TEMP_MA>=1000 AND TEMP_MA<10000 THEN
										sSendString:=CONCAT('FLM',UINT_TO_STRING(TEMP_MA));
									ELSIF TEMP_MA>=100 AND TEMP_MA<1000 THEN
										sSendString:=CONCAT('FLM',UINT_TO_STRING(TEMP_MA));
									ELSIF TEMP_MA>=10 AND TEMP_MA<100 THEN
										sSendString:=CONCAT('FLM0',UINT_TO_STRING(TEMP_MA));
									ELSIF TEMP_MA>=1 AND TEMP_MA<10 THEN
										sSendString:=CONCAT('FLM00',UINT_TO_STRING(TEMP_MA));
									ELSE
										sSendString:='NULL';
									END_IF
									bSend:=BLINK1.OUT;
								
									IF sRecvStringA0=sSendString THEN
										Standby_Step:=60;
									END_IF
									
									TON_MA(IN:=(sRecvStringA0<>sSendString) , PT:=T#5S , Q=> , ET=> );
									IF TON_MA.Q THEN
										WorkStation_TCP.PLC_SEND1.m_nExpStates	:=5;	//参数写入错误
									END_IF				

								60://收到透视信号，跳转到射线阶段
									bSend:=FALSE;
									GVL_State.bScoutSecond:=FALSE;//FUWEI
									IF Entity_IO.bXaryOne THEN
										Standby_Step:=66;
									END_IF;	
									
									sSendString:='ST';		//当前电流
									bSend:=BLINK1_ST.OUT;	//2秒查询一次	
									WorkStation_TCP.PLC_SEND1.m_nExpStates	:=6; 			//参数写入正确
								66:
									TON_DELAY(IN:=FALSE );
									WorkStation_TCP.PLC_SEND1.m_nExpStates	:=7; 			//参数写入后赋其他值
									bSend:=FALSE;
									Main_Step:=30;	
								ELSE
									;
								END_CASE
							END_IF;
						END_IF;
						
						(*-----------------------------------------ER故障无需软件恢复-------------------------------------------------------*)
						IF (sRecvByte[0]= 16#45 AND sRecvByte[1]= 16#52)   THEN //收到ER，只显示故障码，不发送  //16#52  52是ER
							(*处理故障代码显示*)
							CASE RecvNum OF //最多3位故障代码
								3:
									ASCII_Chart_N_Alarm[0](byASCII:=sRecvByte[2] , sOut_Single=> );
									iAlarmNum:=STRING_TO_BYTE(ASCII_Chart_N_Alarm[0].sOut_Single);
								4:
									ASCII_Chart_N_Alarm[1](byASCII:=sRecvByte[2] , sOut_Single=> );
									ASCII_Chart_N_Alarm[2](byASCII:=sRecvByte[3] , sOut_Single=> );
									iAlarmNum:=STRING_TO_BYTE(ASCII_Chart_N_Alarm[1].sOut_Single)*10+STRING_TO_BYTE(ASCII_Chart_N_Alarm[2].sOut_Single);
								5:
									ASCII_Chart_N_Alarm[3](byASCII:=sRecvByte[2] , sOut_Single=> );
									ASCII_Chart_N_Alarm[4](byASCII:=sRecvByte[3] , sOut_Single=> );
									ASCII_Chart_N_Alarm[5](byASCII:=sRecvByte[4] , sOut_Single=> );
									iAlarmNum:=STRING_TO_BYTE(ASCII_Chart_N_Alarm[3].sOut_Single)*100+STRING_TO_BYTE(ASCII_Chart_N_Alarm[4].sOut_Single)*10+STRING_TO_BYTE(ASCII_Chart_N_Alarm[5].sOut_Single);
								ELSE
									iAlarmNum:=iAlarmNum;
							END_CASE	
						END_IF;
							
				30:(*射线准备，出射线阶段*)
					Standby_Step:=0;
					IF (sRecvByte[0]= 16#45 AND sRecvByte[1]= 16#4C) OR sRecvStringA0='ST008' THEN //收到ER或EL,确认收到了错误信号，ER可以理解为可恢复，EL为不可恢复 收到EL信号可复位，ER信号只是显示
						Main_Step:=40;	
					ELSE
						iAlarmNum:=0;//复位故障
						//查询球管热量
						IF sRecvByte[0]=16#48 AND sRecvByte[1]=16#45 THEN //HE 球管热量
							ASCII_Chart_N2[0](byASCII:= sRecvByte[2], sOut_Single=> );
							ASCII_Chart_N2[1](byASCII:= sRecvByte[3], sOut_Single=> );
							ASCII_Chart_N2[2](byASCII:= sRecvByte[4], sOut_Single=> );
							Feedback_nMHuValue:=STRING_TO_REAL(ASCII_Chart_N2[0].sOut_Single)*100+STRING_TO_REAL(ASCII_Chart_N2[1].sOut_Single)*10+STRING_TO_REAL(ASCII_Chart_N2[2].sOut_Single);
						END_IF
						
						IF GVL_State.iPLC_State=40 AND GVL_State.bBooting THEN
							Main_Step		:=20; 				//系统待机下回到射线源待机状态
							Standby_Step	:=10;
							Rad_Step		:=0;
							GVL_State.bBooting:=FALSE;
						ELSE
							(*---------------------------曝光状态---------------------------------*)
							CASE Rad_Step OF
								0://初始化阶段
									TON_DELAY(IN:=FALSE);
									TON_ST(IN:=FALSE);
									Rad_Step:=10;
								10:
									IF sRecvStringA0='FLP1' THEN
										Rad_Step	:=20;
									END_IF;	
									
									IF sRecvStringA0='FLP0' THEN
										Rad_Step	:=40;
									END_IF;	
									
								20://FLX1
									IF sRecvStringA0='FLX1' THEN //OR Entity_IO.bXrayBuckey THEN
										Rad_Step	:=30;
									END_IF;
									
									IF sRecvStringA0='FLP0' THEN
										Rad_Step	:=40;
									END_IF;	
									
								
								30://允许出束阶段
									TON_ST(IN:=FALSE);
									IF sRecvStringA0='FLX0' OR sRecvStringA0='FLP0' THEN //收到FLX0或FLP0，曝光结束
										Rad_Step	:=40;
									ELSE
										;
									END_IF
									
								 40://结束
								 	TON_DELAY(IN:=TRUE , PT:=T#12S , Q=> , ET=> );
									IF TON_DELAY.Q THEN
										Standby_Step:=0;
										Rad_Step	:=88;
										Main_Step	:=20;
									END_IF;
								ELSE
									;
							END_CASE
						END_IF
					END_IF;
					
					(*-----------------------------------------ER故障无需软件恢复-------------------------------------------------------*)
					IF (sRecvByte[0]= 16#45 AND sRecvByte[1]= 16#52)   THEN //收到ER，只显示故障码，不发送  //16#52  52是ER
						(*处理故障代码显示*)
						CASE RecvNum OF //最多3位故障代码
							3:
								ASCII_Chart_N_Alarm[0](byASCII:=sRecvByte[2] , sOut_Single=> );
								iAlarmNum:=STRING_TO_BYTE(ASCII_Chart_N_Alarm[0].sOut_Single);
							4:
								ASCII_Chart_N_Alarm[1](byASCII:=sRecvByte[2] , sOut_Single=> );
								ASCII_Chart_N_Alarm[2](byASCII:=sRecvByte[3] , sOut_Single=> );
								iAlarmNum:=STRING_TO_BYTE(ASCII_Chart_N_Alarm[1].sOut_Single)*10+STRING_TO_BYTE(ASCII_Chart_N_Alarm[2].sOut_Single);
							5:
								ASCII_Chart_N_Alarm[3](byASCII:=sRecvByte[2] , sOut_Single=> );
								ASCII_Chart_N_Alarm[4](byASCII:=sRecvByte[3] , sOut_Single=> );
								ASCII_Chart_N_Alarm[5](byASCII:=sRecvByte[4] , sOut_Single=> );
								iAlarmNum:=STRING_TO_BYTE(ASCII_Chart_N_Alarm[3].sOut_Single)*100+STRING_TO_BYTE(ASCII_Chart_N_Alarm[4].sOut_Single)*10+STRING_TO_BYTE(ASCII_Chart_N_Alarm[5].sOut_Single);
							ELSE
								iAlarmNum:=iAlarmNum;
						END_CASE	
					END_IF;
						
				40:	//错误状态下只显示EL故障
					IF (sRecvByte[0]= 16#45 AND sRecvByte[1]= 16#4C) OR sRecvStringA0='ST008'  THEN 	//收到ER或EL,确认收到了错误信号，ER可以理解为可恢复，EL为不可恢复 收到EL信号可复位，ER信号只是显示
						IF sRecvStringA0='ST008' THEN
							sSendString:='EL ？';
							bSend:=BLINK1.OUT;
						END_IF 
							
						IF Read_0.xDone AND (sRecvByte[0]= 16#45 AND sRecvByte[1]= 16#4C) THEN
							sSendString:=sRecvStringA0;							//收到EL，发送故障码，同时发送EL恢复故障
							f10(CLK:=(sRecvByte[0]= 16#45 AND sRecvByte[1]= 16#4C) AND Read_0.xDone  , Q=> bSend);//发一次回一次
						ELSE
							f10(CLK:=FALSE  , Q=> bSend);//发一次回一次
						END_IF;
						
						BLINK2(ENABLE:=TRUE , TIMELOW:=T#1S , TIMEHIGH:=T#1S , OUT=> );
						IF BLINK2.OUT THEN
							sSendString:='ST';//查询ST状态
							bSend:=BLINK2.OUT AND NOT(f10.Q);
						END_IF
					
						(*处理EL故障代码显示*)
						CASE RecvNum OF //最多3位故障代码
							3:
								ASCII_Chart_N_Alarm[0](byASCII:=sRecvByte[2] , sOut_Single=> );
								iAlarmNum:=STRING_TO_BYTE(ASCII_Chart_N_Alarm[0].sOut_Single);
							4:
								ASCII_Chart_N_Alarm[1](byASCII:=sRecvByte[2] , sOut_Single=> );
								ASCII_Chart_N_Alarm[2](byASCII:=sRecvByte[3] , sOut_Single=> );
								iAlarmNum:=STRING_TO_BYTE(ASCII_Chart_N_Alarm[1].sOut_Single)*10+STRING_TO_BYTE(ASCII_Chart_N_Alarm[2].sOut_Single);
							5:
								ASCII_Chart_N_Alarm[3](byASCII:=sRecvByte[2] , sOut_Single=> );
								ASCII_Chart_N_Alarm[4](byASCII:=sRecvByte[3] , sOut_Single=> );
								ASCII_Chart_N_Alarm[5](byASCII:=sRecvByte[4] , sOut_Single=> );
								iAlarmNum:=STRING_TO_BYTE(ASCII_Chart_N_Alarm[3].sOut_Single)*100+STRING_TO_BYTE(ASCII_Chart_N_Alarm[4].sOut_Single)*10+STRING_TO_BYTE(ASCII_Chart_N_Alarm[5].sOut_Single);
							ELSE
								iAlarmNum:=iAlarmNum;
						END_CASE
						TON40(IN:=FALSE);
					ELSE
						TON40(IN:=TRUE , PT:= T#2S, Q=> , ET=> );
						IF TON40.Q THEN
							Main_Step	:=20;
						END_IF;
					END_IF
				END_CASE
				
*)
END_ACTION

END_PROGRAM

// Device/Application/IOs/Entity_IO
PROGRAM Entity_IO
VAR
	(*0.MC508本体IO,16DI@16DO*)
	//12路200KHz/4路1KHz
	DIB0 AT %IX0.0:BOOL;	DIB1 AT %IX0.1:BOOL;	DIB2 AT %IX0.2:BOOL;	DIB3 AT %IX0.3:BOOL;
	DIB4 AT %IX0.4:BOOL;	DIB5 AT %IX0.5:BOOL;	DIB6 AT %IX0.6:BOOL;	DIB7 AT %IX0.7:BOOL;
	DIB8 AT %IX1.0:BOOL;	DIB9 AT %IX1.1:BOOL;	DIB10 AT %IX1.2:BOOL;	DIB11 AT %IX1.3:BOOL;
	DIB12 AT %IX1.4:BOOL;	DIB13 AT %IX1.5:BOOL;	DIB14 AT %IX1.6:BOOL;	DIB15 AT %IX1.7:BOOL;
	//12路200KHz/4路10KHz
	DOB0 AT %QX0.0:BOOL;	DOB1 AT %QX0.1:BOOL;	DOB2 AT %QX0.2:BOOL;	DOB3 AT %QX0.3:BOOL;
	DOB4 AT %QX0.4:BOOL;	DOB5 AT %QX0.5:BOOL;	DOB6 AT %QX0.6:BOOL;	DOB7 AT %QX0.7:BOOL;
	DOB8 AT %QX1.0:BOOL;	DOB9 AT %QX1.1:BOOL;	DOB10 AT %QX1.2:BOOL;	DOB11 AT %QX1.3:BOOL;
	DOB12 AT %QX1.4:BOOL;	DOB13 AT %QX1.5:BOOL;	DOB14 AT %QX1.6:BOOL;	DOB15 AT %QX1.7:BOOL;
	
	(*1.PM3200 32路DI输入*)
	DIX0 AT %IX4.0:BOOL;DIX1 AT %IX4.1:BOOL;DIX2 AT %IX4.2:BOOL;DIX3 AT %IX4.3:BOOL;
	DIX4 AT %IX4.4:BOOL;DIX5 AT %IX4.5:BOOL;DIX6 AT %IX4.6:BOOL;DIX7 AT %IX4.7:BOOL;
	DIX8 AT %IX5.0:BOOL;DIX9 AT %IX5.1:BOOL;DIX10 AT %IX5.2:BOOL;DIX11 AT %IX5.3:BOOL;
	DIX12 AT %IX5.4:BOOL;DIX13 AT %IX5.5:BOOL;DIX14 AT %IX5.6:BOOL;DIX15 AT %IX5.7:BOOL;
	DIX16 AT %IX6.0:BOOL;DIX17 AT %IX6.1:BOOL;DIX18 AT %IX6.2:BOOL;DIX19 AT %IX6.3:BOOL;
	DIX20 AT %IX6.4:BOOL;DIX21 AT %IX6.5:BOOL;DIX22 AT %IX6.6:BOOL;DIX23 AT %IX6.7:BOOL;
	DIX24 AT %IX7.0:BOOL;DIX25 AT %IX7.1:BOOL;DIX26 AT %IX7.2:BOOL;DIX27 AT %IX7.3:BOOL;
	DIX28 AT %IX7.4:BOOL;DIX29 AT %IX7.5:BOOL;DIX30 AT %IX7.6:BOOL;DIX31 AT %IX7.7:BOOL;
	
	(*2.PM0016-R 16路开关量输出*)
	DOX0 AT %QX2.0:BOOL;DOX1 AT %QX2.1:BOOL;DOX2 AT %QX2.2:BOOL;DOX3 AT %QX2.3:BOOL;
	DOX4 AT %QX2.4:BOOL;DOX5 AT %QX2.5:BOOL;DOX6 AT %QX2.6:BOOL;DOX7 AT %QX2.7:BOOL;
	DOX8 AT %QX3.0:BOOL;DOX9 AT %QX3.1:BOOL;DOX10 AT %QX3.2:BOOL;DOX11 AT %QX3.3:BOOL;
	DOX12 AT %QX3.4:BOOL;DOX13 AT %QX3.5:BOOL;DOX14 AT %QX3.6:BOOL;DOX15 AT %QX3.7:BOOL;
	
	(*3.PM-A0400-IV扩展模块AI*)
	AIX0 AT %IW6:INT;		AIX1 AT %IW7:INT;		AIX2 AT %IW8:INT;		AIX3 AT %IW9:INT;
	
	(*4.内部变量*)
	count: BYTE;
	AIX0_TEMP:INT;
	LS_Counter_0,LS_Counter_1			:LS_Counter;  	//计数器指令实例化
	LS_PresetValue_0,LS_PresetValue_1	:LS_PresetValue;//计数器预设值
	bCalibrate:BOOL;//升降电机标定
	rZeroPos_TEMP:INT;

END_VAR

VAR_INPUT
	bLeftPannel_LED1,bLeftPannel_LED2,bRightPannel_LED1,bRightPannel_LED2: BOOL;//LED灯
	bXaryOne,bXaryTwo,bXaryFlu:BOOL;//X射线一档二档信号
	bLaserOut:BOOL;					//激光灯控制
	bTriggerOut:BOOL;				//射线源Trigger信号
	bUpMotorPos,bUpMotorNeg:BOOL;	//升降电机上升下降控制
	bDelayPower:BOOL;				//延迟断电继电器输出
	bLightYellow:BOOL;				//出束黄色指示灯控制
	bXraySwitch:BOOL;			//触发信号切换继电器/仅在CBCT摸下是PF触发，赋值逻辑也在CBCT里	
	bEmergencyOut:BOOL;
END_VAR

VAR_OUTPUT	
	(*左右面板输入*)
	LeftPannel_BedUp,LeftPannel_BedDown,LeftPannel_BedFore,LeftPannel_BedBack,LeftPannel_LaserButton,LeftPannel_DistanceMove,LeftPannel_RecordPos,LeftPannel_MoveRecordPos: BOOL;
	RightPannel_BedUp,RightPannel_BedDown,RightPannel_BedFore,RightPannel_BedBack,RightPannel_LaserButton,RightPannel_DistanceMove,RightPannel_RecordPos,RightPannel_MoveRecordPos: BOOL;
	(*前进电机和旋转电机限位*)
	bForeMotorMin,bForeMotorMax,bRotateMotorMin,bRotateMotorMax,bUpMotorMin,bUpMotorSTO: BOOL;
	
	bXrayOneInput,bXrayTwoInput,bXrayFluInput,bXayExpoInput:BOOL;
	(*急停和门连锁及钥匙开关*)
	bEmergencyStop,bDoorLock,bKeySwitch,bXzMotorSTO:BOOL;
	
	(*PLC本体输入*)
	iEncoderPulse,iEncoderZ:DINT;(*编码器脉冲信号，4倍频率*)
	rRealPos		:REAL;//升降电机位置实际数值

	bXrayExp:BOOL;
	bSync_out:BOOL;//平板探测器sync_out信号
END_VAR

(*----------------------README--------------------*)
(*PLC功能管脚分配*)

(*0.心跳*)
	count:=count+1;

(*1.左和右PANNEL面板输入*)
	LeftPannel_BedUp		:=DIX3;//床升
	LeftPannel_BedDown		:=DIX4;//床降
	LeftPannel_BedFore		:=DIX5;//床进
	LeftPannel_BedBack		:=DIX2;//床出
	LeftPannel_LaserButton	:=DIX1;//激光灯开关 
	LeftPannel_DistanceMove	:=DIX7;//固定距离进床 ,修改为一键0°
	LeftPannel_RecordPos	:=DIX0;//记录预设位置
	LeftPannel_MoveRecordPos:=DIX6;//运动到预设位置
	
	RightPannel_BedUp		:=DIX11;//床升     
	RightPannel_BedDown		:=DIX12;//床降     
	RightPannel_BedFore		:=DIX13;//床进     
	RightPannel_BedBack		:=DIX10;//床出     
	RightPannel_LaserButton	:=DIX15;//激光灯开关  
	RightPannel_DistanceMove:=DIX9; //固定距离进床 修改为一键0°
	RightPannel_RecordPos	:=DIX14;//记录预设位置 
	RightPannel_MoveRecordPos:=DIX8; //运动到预设位置,
	
(*2.Pannel面板指示灯，左下角D10是LED1,右下角D11是LED2*)
	DOB0:=bTriggerOut	;		//射线源触发信号
	
	DOB8:=bLeftPannel_LED1;		//左面板LED1灯，对应激光灯按钮
	DOB9:=bLeftPannel_LED2;		//左面板LED2灯，对应固定距离进床
	DOB10:=bRightPannel_LED1;	//右面板LED1灯，对应固定距离进床
	DOB11:=bRightPannel_LED2;	//右面板LED2灯，对应激光灯按钮


(*3.限位信号及急停门连锁信号*)
	(*以下4个限位信号只能接入驱动器，不支持同时接入PLC，PLC获取开关信息从PDO中获得*)
	bForeMotorMin	:=bForeMotorMin1;//前进电机最小限位
	bForeMotorMax	:=bForeMotorMax1;//前进电机最大限位
	bRotateMotorMin	:=bRotateMotorMin1;//旋转电机最小限位DI1-
	bRotateMotorMax	:=bRotateMotorMax1;//旋转电机最大限位DI2-
	
//	bUpMotorMin		:=NOT(DIX16);//升降电机下限位，下限位信号
bUpMotorMin	:=FALSE;
	bUpMotorSTO		:=DIX17;//前进电机电机STO反馈
	bXrayOneInput 	:=(DIX18);
	bXrayTwoInput 	:=(DIX19);
	bXayExpoInput 	:=(DIX20); 
	bXrayFluInput 	:=(DIX21);
	
	
	bKeySwitch		:=DIX24;//钥匙开关开机信号
	bDoorLock		:=DIX25;//门连锁信号
	bEmergencyStop	:=NOT(DIX26);//急停停止信号
	bXzMotorSTO		:=DIX27;//旋转电机STO反馈

(*4.PLC本体输入*)
	
(*5.编码器信号输入，4倍频率*)
	LS_Counter_0(xEnable:=TRUE , eChannel:= 4 , xValid=> , xError=> , eErrorID=> , diValue=>iEncoderPulse );
	LS_Counter_1(xEnable:=TRUE , eChannel:= 5 , xValid=> , xError=> , eErrorID=> , diValue=>iEncoderZ );

(*6.模拟量采集输入*)
	IF AIX0<=0 THEN
		AIX0_TEMP:=0;
	ELSIF AIX0>=32000 THEN
		AIX0_TEMP:=32000;
	ELSE
		AIX0_TEMP:=AIX0;
	END_IF

	(*6.1.标定*)
	IF bCalibrate THEN 
		GVL_Retain.rSJ_Zero:=LIMIT(0 ,AIX0_TEMP ,32000);
	//	bCalibrate:=FALSE;
	END_IF
	
	(*6.2.计算实际高度*)
	rRealPos:=400*INT_TO_REAL(AIX0-GVL_Retain.rSJ_Zero)/32000;
	
(*7.开关量输出管脚分配*)
	DOX0:= bUpMotorPos		;		//电机上升控制
	DOX1 :=	bUpMotorNeg		;		//电机下降控制
	DOX2 :=	bXraySwitch		;		//射线源切换触发方式继电器
						
	DOX4 :=	bLightYellow	;		//出束黄色指示灯控制
	DOX5 :=	bLaserOut	  	;		//激光灯输出
	DOX6 :=	bEmergencyOut	;		//软件急停
						
	DOX8 :=	bDelayPower		;		//延迟断电继电器控制
	DOX12:=	bXaryOne	   	;		//X射线一档输出信号
	DOX13:=	bXaryTwo	   	;		//X射线二档输出信号
	DOX14:=	bXaryFlu	   	;		//X射线透视输出信号

		
	bXrayExp:=DIB7;
	bSync_out:=DIX31;//探测器sync_out 输出

END_PROGRAM

// Device/Application/Communication/CTBOX_RS232
PROGRAM CTBOX_RS232
VAR
	Open_0: COM.Open;
	Write_0: COM.Write;
	Read_0: COM.Read;
	Close_0: COM.Close;
	xOpen_Exe:BOOL;
	hComHandle:CAA.HANDLE;
	byWriteData:ARRAY [0..12] OF BYTE;
	xWrite_Exe:BOOL;
	xRead_Exe:BOOL;
    byReadData:ARRAY [0..15] OF BYTE;
    xClose_Exe:BOOL;
	aParamsB19200 : ARRAY [1..7] OF COM.PARAMETER := [
    (udiParameterId := COM.CAA_Parameter_Constants.udiPort,udiValue := 4), 					//指令端口2,3,4,5分别对应硬件接口com2、com0、com1、com3
    (udiParameterId := COM.CAA_Parameter_Constants.udiBaudrate,udiValue := 19200),			//波特率，设置为19200
    (udiParameterId := COM.CAA_Parameter_Constants.udiParity,udiValue := COM.PARITY.NONE),	//校验，设置为无校验
    (udiParameterId := COM.CAA_Parameter_Constants.udiStopBits,udiValue := COM.STOPBIT.ONESTOPBIT),//停止位，1位
    (udiParameterId := COM.CAA_Parameter_Constants.udiTimeout,udiValue := 500),				//超时时间，设置成500ms
    (udiParameterId := COM.CAA_Parameter_Constants.udiByteSize,udiValue := 8),				//数据位
    (udiParameterId := COM.CAA_Parameter_Constants.udiBinary, udiValue := 1)				//二进制参数，启用二进制模式
];		
	Check:UINT;//读取数据的和校验
	TON1,TON2:TON;//定时写入和读取数据
	TON3:Standard.TON;//延时打开串口
	TON_Reset:Standard.TON;
	i: INT;//
	CTBOX_KEY	:ARRAY [0..7] OF BOOL;
	Blink_Reset:Blink;
	Lamp5State,Lamp6State,Lamp7State,Lamp8State:BYTE;
	
	count: BYTE;
	bDebug_RS232:BOOL;
	A1,A2,A3,A4:BOOL;
	R_CLOSE:Standard.R_TRIG;
	bReset:BOOL;
	booting:BOOL:=TRUE;
	R_TRIG11:R_TRIG;
	
	TOF_Delay:ARRAY [0..7] OF Standard.TOF;
	
	SampleBooleanCheck1:ARRAY [0..7] OF SampleBooleanCheck;
END_VAR

VAR_OUTPUT
	CTBOX_KEY_Manual		:BOOL;//手动扫描
	CTBOX_KEY_Auto			:BOOL;//自动扫描
	CTBOX_KEY_Stop			:BOOL;//中止扫描
	CTBOX_KEY_MoveDistance	:BOOL;//移动到扫描位置
	CTBOX_KEY_BedFore		:BOOL; //进床
	CTBOX_KEY_BedUp			:BOOL;//升床
	CTBOX_KEY_BedBack		:BOOL;//出床
	CTBOX_KEY_BedDown		:BOOL;//升床	
END_VAR

(*Readme*)
(*与CTbox进行通信*)
(*------------------------------------第一部分：RS232数据收发设置---------------------------------------*)
(*0.心跳*)
	IF R_TRIG11.Q THEN
		count:=count+1;
	END_IF;
	R_TRIG11(CLK:=Write_0.xDone , Q=> );
(*1.open*)
	IF booting AND TON3.Q  THEN
		bReset:=TRUE;
		booting:=FALSE;
	END_IF
	
	TON3(IN:=TRUE , PT:=T#10S);//开机后10秒打开串口
	Open_0(xExecute:=bReset , xDone=> , xBusy=> , xError=> , usiListLength:=20 , pParameterList:=ADR(aParamsB19200) , eError=> , hCom=>hComHandle );
	
(*2.Write*)
	TON1(IN:=NOT TON1.Q , PT:=T#58MS , Q=> , ET=> );
	Write_0(
			xExecute:= Open_0.xDone AND TON1.Q, //周期写入控制灯的命令，同时此命令也是查询CTBOX键值的命令，主动发才会回复键值
			xAbort:= , 
			udiTimeOut:=500 , 
			xDone=> , 
			xBusy=> , 
			xError=> , 
			xAborted=> , 
			hCom:= hComHandle, 
			pBuffer:= ADR(byWriteData), 
			szSize:= 12, 
			eError=> );	
	
		byWriteData[0]:=16#FD;
		byWriteData[1]:=16#F4;
		byWriteData[2]:=16#03;
		byWriteData[3]:=16#04;
		
		byWriteData[4]:=16+Lamp7State;
		byWriteData[5]:=32+Lamp8State;
		byWriteData[6]:=48+Lamp6State;
		byWriteData[7]:=64+Lamp5State;
		
		Check:=USINT_TO_UINT(byWriteData[0])+USINT_TO_UINT(byWriteData[1])+USINT_TO_UINT(byWriteData[2])+USINT_TO_UINT(byWriteData[3])+
					USINT_TO_UINT(byWriteData[4])+USINT_TO_UINT(byWriteData[5])+USINT_TO_UINT(byWriteData[6])+USINT_TO_UINT(byWriteData[7]);
		byWriteData[8]:=UINT_TO_USINT(Check MOD 256);   
		byWriteData[9]:=UINT_TO_USINT(Check / 256);
		byWriteData[10]:=16#4F;
		byWriteData[11]:=16#DF;
		
(*3.Read*)
	TON2(IN:=NOT TON2.Q , PT:=T#36MS , Q=> , ET=> );
	Read_0(
			xExecute:= Open_0.xDone AND TON2.Q AND NOT(xWrite_Exe), 
			xAbort:= , 
			udiTimeOut:= 500, 
			xDone=> , 
			xBusy=> , 
			xError=> , 
			xAborted=> , 
			hCom:= hComHandle, 
			pBuffer:= ADR(byReadData), 
			szBuffer:= 16, 
			eError=> , 
			szSize=> );
	
(*4.Close*)
	Close_0(
			xExecute:= xClose_Exe, 
			xDone=> , 
			xBusy=> , 
			xError=> , 
			hCom:= hComHandle, 
			eError=> );
			
(*5.Reset*)
(*	IF TON3.Q THEN			//开机10秒后在进行开始故障复位逻辑
		TON_Reset(IN:=(Read_0.szSize=0), PT:=T#2S , Q=> , ET=> ); 
		Blink_Reset(ENABLE:=TON_Reset.Q, TIMELOW:=T#5S , TIMEHIGH:=T#20MS , OUT=> );
		R_CLOSE(CLK:= TON_Reset.Q AND Blink_Reset.OUT, Q=> xClose_Exe);
		IF TON_Reset.Q AND Close_0.xDone THEN
			bReset:=TON_Reset.Q AND NOT(Blink_Reset.OUT);
		ELSE
			bReset:=TRUE;
		END_IF;
	END_IF			
*)		
(*---------------------------第二部分：数据处理---------------------------*)
(*2.1 数据接收处理*)
	IF byReadData[0]=16#FD AND byReadData[1]=16#F4 AND byReadData[2]=16#2 AND byReadData[3]=16#08 
		AND byReadData[14]=16#4F AND byReadData[15]=16#DF THEN	
		FOR i:=0 TO 7 BY 1 DO
			CTBOX_KEY[i]:=BYTE_TO_BOOL(byReadData[i+4]);
		END_FOR
	ELSE
		FOR i:=0 TO 7 BY 1 DO
    		CTBOX_KEY[i]:=FALSE;
		END_FOR
	END_IF
	
	FOR i:=0 TO 7 BY 1 DO
		SampleBooleanCheck1[i](bSampleInput:=CTBOX_KEY[i] , NumX:= 40, Num:=10 , bFinalOutput=> );
	END_FOR
	
(*2.2.管脚分配*)	
	CTBOX_KEY_Manual		:=SampleBooleanCheck1[0].bFinalOutput;    
	CTBOX_KEY_Auto			:=SampleBooleanCheck1[1].bFinalOutput;    		      
	CTBOX_KEY_Stop			:=SampleBooleanCheck1[2].bFinalOutput;    	      
	CTBOX_KEY_MoveDistance	:=SampleBooleanCheck1[3].bFinalOutput;    
	CTBOX_KEY_BedFore		:=SampleBooleanCheck1[4].bFinalOutput  ;    
	CTBOX_KEY_BedUp			:=SampleBooleanCheck1[5].bFinalOutput;     
	CTBOX_KEY_BedBack		:=SampleBooleanCheck1[6].bFinalOutput ;     
	CTBOX_KEY_BedDown		:=SampleBooleanCheck1[7].bFinalOutput;  


(*3 数据发送处理*)
(*------5678四个灯状态处理-------------*)
	IF WorkMode.iWorkMode=99 AND bDebug_RS232 THEN		
		IF A1 THEN
			A2:=FALSE;
			A3:=FALSE;
			A4:=FALSE;
			Lamp5State:=16#00;
			Lamp6State:=16#00;
			Lamp7State:=16#00;
			Lamp8State:=16#00;
		ELSE
			IF A2 THEN
				A3:=FALSE;
				A4:=FALSE;
				Lamp5State:=16#02;
				Lamp6State:=16#02;
				Lamp7State:=16#02;
				Lamp8State:=16#02;
			ELSE
				IF A3 THEN
					A4:=FALSE;
					Lamp5State:=16#03;
					Lamp6State:=16#03;
					Lamp7State:=16#03;
					Lamp8State:=16#03;
				ELSE
					IF A4 THEN
						Lamp5State:=16#01;
						Lamp6State:=16#01;
						Lamp7State:=16#01;
						Lamp8State:=16#01;
					ELSE
						Lamp5State:=16#00;
						Lamp6State:=16#00;
						Lamp7State:=16#00;
						Lamp8State:=16#00;
					END_IF
				END_IF
			END_IF
		END_IF
	ELSE  //正常工作流程下的处理
		CASE PLC_PRG.LampCmd5 OF 
			E_LampCmd.关闭:Lamp5State:=16#00;
			E_LampCmd.常亮:Lamp5State:=16#01;
			E_LampCmd.慢闪:Lamp5State:=16#02;
			E_LampCmd.快闪:Lamp5State:=16#03;
			ELSE Lamp5State:=16#00;
		END_CASE
		
		CASE PLC_PRG.LampCmd6 OF 
			E_LampCmd.关闭:Lamp6State:=16#00;
			E_LampCmd.常亮:Lamp6State:=16#01;
			E_LampCmd.慢闪:Lamp6State:=16#02;
			E_LampCmd.快闪:Lamp6State:=16#03;
			ELSE Lamp6State:=16#00;
		END_CASE
		
			CASE PLC_PRG.LampCmd7 OF 
			E_LampCmd.关闭:Lamp7State:=16#00;
			E_LampCmd.常亮:Lamp7State:=16#01;
			E_LampCmd.慢闪:Lamp7State:=16#02;
			E_LampCmd.快闪:Lamp7State:=16#03;
			ELSE Lamp7State:=16#00;
		END_CASE
		
		CASE PLC_PRG.LampCmd8 OF 
			E_LampCmd.关闭:Lamp8State:=16#00;
			E_LampCmd.常亮:Lamp8State:=16#01;
			E_LampCmd.慢闪:Lamp8State:=16#02;
			E_LampCmd.快闪:Lamp8State:=16#03;
			ELSE Lamp8State:=16#00;
		END_CASE
	END_IF;

END_PROGRAM

// Device/Application/Logic/WorkMode
PROGRAM WorkMode
VAR
	count	:BYTE;	
	WorkModeTemp:INT:=99;//默认
	TON1,TON2	:TON;
	bDebugMode	:BOOL:=FALSE;
	booting:BOOL	:=TRUE;
END_VAR

VAR_OUTPUT	
	iWorkMode	:INT;
END_VAR

(*Readme*)
	(*0.心跳*)
	count:=count+1;
	TON1(IN:= TRUE, PT:= T#10S, Q=> , ET=> );
	(*状态机切换逻辑，再复杂的话用if-condition方式*)
	IF (Entity_IO.bKeySwitch=FALSE) AND TON1.Q THEN			//记着取消NOT
		WorkModeTemp:=55;									//55 关机模式
		booting:=TRUE;
	ELSE
		IF bDebugMode THEN
			WorkModeTemp:=99;						//调试模式
		ELSE
			IF (Entity_IO.bEmergencyStop) THEN		//TRUE相当于被触发了
				WorkModeTemp:=33;					//急停模式
			ELSE
				IF Axis_XZ.XZ_AxisState.bAxisErr OR Axis_QJ.QJ_AxisState.bAxisErr OR Axis_XZ.XZ_AxisState.bErrStop OR  Axis_QJ.QJ_AxisState.bErrStop THEN
					WorkModeTemp:=44;				//错误模式
				ELSE
					WorkModeTemp:=11;				//工作状态
				END_IF
			END_IF
		END_IF
	END_IF

	iWorkMode:=	WorkModeTemp;//44,11,99

END_PROGRAM

// Device/Application/BasicFBs/SampleBooleanCheck
FUNCTION_BLOCK SampleBooleanCheck
VAR_INPUT
	 // 待采样的布尔型变量（可外接传感器/其他信号）
    bSampleInput: BOOL;
	NumX:INT;
	Num:INT;
END_VAR
VAR_OUTPUT
	 // 最终输出结果
    bFinalOutput: BOOL ;
END_VAR
VAR
	// TRUE结果的累计计数器
    nTrueCount: INT := 0;
    // 采样触发信号（例如定时器、外部触发脉冲）
    bSampleTrigger: BOOL:=TRUE;
	nSampleCount: INT:=0 ; // 采样次数计数器（记录已完成的采样次数）
END_VAR

// 核心采样逻辑：每次触发采样时执行
    // 仅在采样次数未达到10次时执行采样
		IF nSampleCount < NumX THEN
			// 采样次数+1
			nSampleCount := nSampleCount + 1;
			// 如果当前采样值为TRUE，累计TRUE次数
			IF bSampleInput THEN
				nTrueCount := nTrueCount + 1;
			END_IF;
			
			// 当完成10次采样后，判断结果
			IF nSampleCount >= NumX THEN
				// 5次及以上为TRUE则输出TRUE，否则FALSE
				bFinalOutput := nTrueCount >= Num;
				// 重置计数器，为下一轮10次采样做准备
				nSampleCount := 0;
				nTrueCount := 0;
			END_IF;
		ELSE
			nSampleCount := 0;
			nTrueCount := 0;
		END_IF;

END_FUNCTION_BLOCK

// Device/Application/Motor/Motor_SJ
PROGRAM Motor_SJ
VAR
	count		:BYTE;
	Mode		:INT;
	DB:REAL		:=15;
	R_TRIG1,R_TRIG2	:R_TRIG;
	bMovPos:BOOL;
END_VAR

VAR_INPUT
	Enable:BOOL;
END_VAR

VAR_OUTPUT	
//	rRealPos:REAL;
END_VAR

(*-----------------------------Readme---------------------------------*)
(*---------升降电机功能块---------------------------------------------*)
(*-------------输入管脚已有滤波-------------------710-920-----------700-930----*)


(*0.心跳*)
	count:=count+1;
	
(*3.点动及位置控制，如果触碰到限位，首先手动移动到安全区域*)
	IF Enable THEN
		(*1.同时按了上升和下降*)
		IF (Entity_IO.LeftPannel_BedUp OR Entity_IO.RightPannel_BedUp OR CTBOX_RS232.CTBOX_KEY_BedUp) 
				AND (Entity_IO.LeftPannel_BedDown OR Entity_IO.RightPannel_BedDown OR CTBOX_RS232.CTBOX_KEY_BedDown) THEN
			Mode:=0;
			bMovPos:=FALSE;
		(*2.上升*)
		ELSIF (Entity_IO.LeftPannel_BedUp OR Entity_IO.RightPannel_BedUp OR CTBOX_RS232.CTBOX_KEY_BedUp)=TRUE 
				AND (Entity_IO.LeftPannel_BedDown=FALSE AND Entity_IO.RightPannel_BedDown=FALSE AND CTBOX_RS232.CTBOX_KEY_BedDown=FALSE) THEN
			bMovPos:=FALSE;
			IF Entity_IO.rRealPos<=210 THEN
				Mode:=10;
			ELSE
				Mode:=0;
			END_IF
		(*3.下降*)
		ELSIF (Entity_IO.LeftPannel_BedUp=FALSE AND Entity_IO.RightPannel_BedUp=FALSE AND CTBOX_RS232.CTBOX_KEY_BedUp=FALSE) 
			AND (Entity_IO.LeftPannel_BedDown OR Entity_IO.RightPannel_BedDown OR CTBOX_RS232.CTBOX_KEY_BedDown)=TRUE THEN
			bMovPos:=FALSE;
			IF Entity_IO.rRealPos>=0 THEN
				Mode:=20;
			ELSE
				Mode:=0;
			END_IF
		(*4.上升下降都没按*)
		ELSE
			(*位置控制*)
			R_TRIG1(CLK:= Entity_IO.LeftPannel_MoveRecordPos OR Entity_IO.RightPannel_MoveRecordPos, Q=> );
			IF R_TRIG1.Q THEN
				bMovPos:=TRUE;
			END_IF
			
			IF bMovPos THEN
				IF Entity_IO.rRealPos<(GVL_Retain.rBedRecordHeight-DB) THEN
					 Mode:=10;
				ELSIF Entity_IO.rRealPos>(GVL_Retain.rBedRecordHeight+DB)  THEN
					 Mode:=20;
				ELSE
					 Mode:=0;
				END_IF
			ELSE
				 Mode:=0;
			END_IF
		END_IF
	ELSE
		Mode:=0;
	END_IF
	
	
	CASE Mode OF 
	0://禁止运动
		Entity_IO.bUpMotorPos:=FALSE;
		Entity_IO.bUpMotorNeg:=FALSE;
	10://上升
		Entity_IO.bUpMotorPos:=TRUE;
		Entity_IO.bUpMotorNeg:=FALSE;
	20://下降
		Entity_IO.bUpMotorPos:=FALSE;
		Entity_IO.bUpMotorNeg:=TRUE;
	END_CASE

END_PROGRAM

// Device/Application/Init/InitMotor
PROGRAM InitMotor
VAR
	sNameXZ,sNameQJ,sNameSJ: WSTRING:="";
END_VAR

(*Readme*)
(*电机初始化程序*)

(*1.电机名称*)
	sNameXZ:="旋转电机";
	sNameQJ:="前进电机";
	sNameSJ:="升降电机";
	
(*2.电机默认参数设置*)
	Axis_QJ.QJ_AxisCmd.AxisPara.rAbsVelocity:=60;
	Axis_QJ.QJ_AxisCmd.AxisPara.rAccDec:=400;//0117
	Axis_QJ.QJ_AxisCmd.AxisPara.rJogVelocity:=60;
	Axis_QJ.QJ_AxisCmd.AxisPara.rRelVelocity:=30;
	
	Axis_XZ.XZ_AxisCmd.AxisPara.rAbsVelocity:=10;
	Axis_XZ.XZ_AxisCmd.AxisPara.rAccDec:=50;
	Axis_XZ.XZ_AxisCmd.AxisPara.rJogVelocity:=30;
	Axis_XZ.XZ_AxisCmd.AxisPara.rRelVelocity:=30;
	(*回零参数*)
	Axis_XZ.XZ_AxisCmd.AxisPara.rHomeHighSpeed:=30;
	Axis_XZ.XZ_AxisCmd.AxisPara.rHomeLowSpeed:=10;
	Axis_XZ.XZ_AxisCmd.AxisPara.rHomeAcc:=50;
	
	Axis_QJ.QJ_AxisCmd.AxisPara.rHomeHighSpeed:=30;
	Axis_QJ.QJ_AxisCmd.AxisPara.rHomeLowSpeed:=5;
	Axis_QJ.QJ_AxisCmd.AxisPara.rHomeAcc:=5;

END_PROGRAM

// Device/Application/Refer/Trigger_HaoboPannel
PROGRAM Trigger_HaoboPannel
VAR
	count:BYTE;
	booting:BOOL:=TRUE;
	iHopePulse:UINT;
	EncoderNum:UDINT;
	EncoderNum1:DINT;
	iValidTrigger:UINT;
	NumTrigger:BYTE:=4;
	NumTrigger1:BYTE:=28; //DR扫，固定角度曝光28次
	
	TOF_Trig,TOF_Scout:Standard.TOF;
	Blink_Scout:Blink;
	F_TRIG1,F_TRIG2:Standard.F_TRIG;
	R_TRIG1,R_TRIG2:Standard.R_TRIG;
	
	iStartTrigger:UDINT;		//记录开始扫描的起始位置，编码器数值
	iStartTrigger1:DINT;		//记录开始扫描的起始位置，编码器数值
	DB_EncoderNum:UDINT;		//差值
	DB_EncoderNum1:DINT;		//差值
	bTiggerEnable:BOOL;
	R_TRIG_EnableHaobo1,R_TRIG_EnableHaobo2:R_TRIG;
	TON1,TON2:TON;
END_VAR

VAR_INPUT
	iSamplingRate:UINT;
	bEnableTrigger:BOOL;
	bEnableScout:BOOL;
END_VAR

VAR_OUTPUT	
	iActNumPulse:UINT;//有效触发次数
	bScoutPulse:BOOL;
END_VAR

(*README*)
(*脉冲触发信号处理,探测器触发勾选0.Polarity_Param 2.i_HVG_Request 下降沿触发 ，不勾选是上升沿触发*)
(*
(*0.心跳*)
	count:=count+1;
	
(*1.初始化函数*)
	IF booting THEN
		booting:=FALSE;
	END_IF
	
(*2.获取上位机发送的采样率*)//
	iSamplingRate:=UDINT_TO_UINT(WorkStation_TCP.PLC_RECV1.m_nSamplingRate);//采样率，有4个选项：2400帧/圈；1200帧/圈；600帧/圈,360帧/圈 recv[21]
	
(*3.处理多少个脉冲输出一个trigger*)
	CASE iSamplingRate OF 
		360:
			iHopePulse:=360;
		600:
			iHopePulse:=216;
		1200:
			iHopePulse:=108;
		2400:
			iHopePulse:=54;
		ELSE
			iHopePulse:=360;
	END_CASE
	
(*4.获取旋转编码器的数值*)
	EncoderNum1:=Entity_IO.iEncoderPulse;
	
(*6.开启相对位置，记录开始位置*)	
	R_TRIG2(CLK:=GVL_SCAN.bEnableTrigger , Q=> );
	IF R_TRIG2.Q THEN
		iStartTrigger1:=EncoderNum1;
	END_IF
	
(*6.主逻辑，分2个工作模式，1是根据CBCT角度旋转触发，一个是根据定位像连续触发三次，次数可设*)
	TOF_Trig(IN:= GVL_SCAN.bEnableTrigger, PT:=T#1S , Q=> , ET=> 	);	//使能触发
	TOF_Scout(IN:= GVL_SCAN.bEnableScout,  PT:=T#3S , Q=> , ET=> 	);	//定位像自动触发标志
	
	IF GVL_SCAN.bEnableTrigger AND Entity_IO.bXaryOne THEN
		(*---------------------------处理相对脉冲来作为触发--------------------------------------*)
		DB_EncoderNum1:=ABS(EncoderNum1-iStartTrigger1);
		iValidTrigger:=DINT_TO_UINT(DB_EncoderNum1 MOD iHopePulse);
		
		(*--------------------------CBCT扫描，根据角度输出曝光指令-------------------------------*)
		IF GVL_State.iPLC_State=60 THEN
			(*加时间滤波，经分析，发现增量编码器有跳变的情况出现*)
			(*1.10ms判断*)
			TON1(IN:=Entity_IO.bTriggerOut , PT:=T#12MS , Q=> );
			R_TRIG_EnableHaobo1(CLK:=TON1.Q , Q=> );
			R_TRIG_EnableHaobo2(CLK:=Entity_IO.bTriggerOut , Q=> );
			IF R_TRIG_EnableHaobo1.Q THEN
				bTiggerEnable:=TRUE;
			END_IF
			(*2.出射线后才会出图*)
			IF R_TRIG_EnableHaobo2.Q THEN
				bTiggerEnable:=FALSE;
			END_IF
			(*3.正常出射线出图*)
			IF (iActNumPulse)<=(iSamplingRate+2) THEN
				IF (iValidTrigger)<=1*iHopePulse / 3 THEN  //1/3的占空比，这个时间要和上位机下发的扫描时间对应
					Entity_IO.bTriggerOut:=TRUE;
					Entity_IO.bTriggerHaobo:=FALSE;
				ELSE
					Entity_IO.bTriggerOut:=FALSE;
					Entity_IO.bTriggerHaobo:=bTiggerEnable;
				END_IF
			ELSE
				Entity_IO.bTriggerOut:=FALSE;
				Entity_IO.bTriggerHaobo:=FALSE;
			END_IF
			
			(*-----------------------计数器清零操作-----------------------*)
			IF PLC_PRG.Step_CBCT<=70 THEN
				iActNumPulse:=0;
				Entity_IO.bTriggerOut:=FALSE;
				Entity_IO.bTriggerHaobo:=FALSE;
				bTiggerEnable:=FALSE;
			END_IF
		END_IF	
		(*-------------------------定位像扫描，固定角度直接曝光4次--------------------------------*)
		IF GVL_State.iPLC_State=50 THEN
			IF TOF_Scout.Q=TRUE THEN
			(*-----------------三个以内正常输出------曝光4次----------------------*)
				IF iActNumPulse<NumTrigger THEN
					Blink_Scout(ENABLE:= TRUE, TIMELOW:=T#40MS , TIMEHIGH:=T#40MS , OUT=> );	//TIMEHIGH 的时间要小于曝光时间，当前曝光时间是10ms
					Entity_IO.bTriggerOut:=Blink_Scout.OUT;
					Entity_IO.bTriggerHaobo:=NOT(Blink_Scout.OUT);
					bScoutPulse:=TRUE;			//定位像曝光中
				ELSE
					Blink_Scout(ENABLE:= FALSE);
					Entity_IO.bTriggerOut:=FALSE;
					Entity_IO.bTriggerHaobo:=FALSE;
					bScoutPulse:=FALSE;
				END_IF
			ELSE
				Blink_Scout(ENABLE:= FALSE);
				Entity_IO.bTriggerOut:=FALSE;
				Entity_IO.bTriggerHaobo:=FALSE;
				bScoutPulse:=FALSE;
			END_IF
		END_IF
		
		(*-------------------------DR扫描，固定角度直接曝光28次-------------新增DR扫，固定角度曝光33次0616-----------------*)
		IF GVL_State.iPLC_State=55 OR GVL_State.iPLC_State=58 THEN
			IF TOF_Scout.Q=TRUE THEN
			(*-----------------28个以内正常输出------曝光28次----------------------*)
				IF iActNumPulse<NumTrigger1 THEN
					Blink_Scout(ENABLE:= TRUE, TIMELOW:=T#40MS , TIMEHIGH:=T#40MS , OUT=> );	//TIMEHIGH 的时间要小于曝光时间，当前曝光时间是10ms
					Entity_IO.bTriggerOut:=Blink_Scout.OUT;
					Entity_IO.bTriggerHaobo:=NOT(Blink_Scout.OUT);
					bScoutPulse:=TRUE;			//定位像曝光中
				ELSE
					Blink_Scout(ENABLE:= FALSE);
					Entity_IO.bTriggerOut:=FALSE;
					Entity_IO.bTriggerHaobo:=FALSE;
					bScoutPulse:=FALSE;
				END_IF
			ELSE
				Blink_Scout(ENABLE:= FALSE);
				Entity_IO.bTriggerOut:=FALSE;
				Entity_IO.bTriggerHaobo:=FALSE;
				bScoutPulse:=FALSE;
			END_IF
		END_IF
	ELSE
		bTiggerEnable:=FALSE;
		Entity_IO.bTriggerOut:=FALSE;
		Entity_IO.bTriggerHaobo:=FALSE;
	END_IF
	
	(*-----------------计数一共有多少个脉冲输出--------------------*)
	F_TRIG2(CLK:=(Entity_IO.bTriggerHaobo) 
			AND (GVL_State.iPLC_State=50 OR GVL_State.iPLC_State=60 OR GVL_State.iPLC_State=55 OR GVL_State.iPLC_State=65 OR GVL_State.iPLC_State=58) 
			AND (PLC_PRG.Step_Scout<>42 OR PLC_PRG.Step_DR<>42)  , Q=> );
	IF F_TRIG2.Q THEN					(*计数一共输出多少脉冲*)
		iActNumPulse:=iActNumPulse+1;
	END_IF;
	
(*8.计数器清零*)	
	IF GVL_State.iPLC_State=50 THEN
		(*-----------------------计数器清零操作-----------------------*)
		IF PLC_PRG.Step_Scout<=42 OR PLC_PRG.Step_Scout>=70 THEN
			iActNumPulse:=0;
			Entity_IO.bTriggerOut:=FALSE;
			Entity_IO.bTriggerHaobo:=FALSE;
		END_IF
	ELSIF GVL_State.iPLC_State=55 THEN
		IF PLC_PRG.Step_DR<=42 OR PLC_PRG.Step_DR>=70 THEN
			iActNumPulse:=0;
			Entity_IO.bTriggerOut:=FALSE;
			Entity_IO.bTriggerHaobo:=FALSE;
		END_IF
	ELSIF GVL_State.iPLC_State=60 THEN
		(*-----------------------计数器清零操作-----------------------*)
		IF PLC_PRG.Step_CBCT<=70 THEN
			iActNumPulse:=0;
			Entity_IO.bTriggerOut:=FALSE;
			Entity_IO.bTriggerHaobo:=FALSE;
		END_IF
	ELSIF GVL_State.iPLC_State=58 THEN
		(*-----------------------计数器清零操作-----------------------*)
		IF PLC_PRG.Step_AutoDR<=70 THEN
			iActNumPulse:=0;
			Entity_IO.bTriggerOut:=FALSE;
			Entity_IO.bTriggerHaobo:=FALSE;
		END_IF
	ELSIF GVL_State.iPLC_State=40 THEN
		iActNumPulse:=0;
	END_IF
	
*)

END_PROGRAM

// Device/Application/RecordLog/RecordLog
PROGRAM RecordLog
VAR
	(*--------------------------------------------第一部分：文件操作变量-------------------------------------------------------*)
	//ACT_SysFileOpen 变量
    xFileOpen: BOOL := FALSE;  //打开文件使能
	PathName: STRING := '/usr/src/CODESYSControl/UsrData/test1.txt';  //文件路径及文件名
	OpenErrorID: RTS_IEC_RESULT;   //文件打开错误码
	hFile: RTS_IEC_HANDLE := RTS_INVALID_HANDLE;  //文件句柄
//ACT_SysFileClose 变量	
	xFileClose: BOOL := FALSE;   //关闭文件使能
	FileCloseErrorID: RTS_IEC_RESULT;  //文件关闭错误码
//ACT_SysFileCopy 变量	
	xFileCopy: BOOL := FALSE; //复制文件使能
	CoDestFileName: STRING :='/usr/src/CODESYSControl/UsrData/test1_copy.txt' ; //目标文件路径及文件名
	CoSourceFileName: STRING := '/usr/src/CODESYSControl/UsrData/test1.txt';  //源文件路径及文件名
	CoSize: __XWORD := 0;  //实际复制文件大小，单位字节
	FileCopyErrorID: RTS_IEC_RESULT :=0;   //文件复制错误码
//ACT_SysFileDelete 变量
	xFileDelete: BOOL := FALSE;  //删除文件使能
	DelFileName: STRING :='/usr/src/CODESYSControl/UsrData/test1.txt';  //删除的文件路径及文件名
	FileDeleteErrorID: RTS_IEC_RESULT;  //文件删除错误码
//ACT_SysFileRead 变量	
	xFileRead: BOOL := FALSE;   //读取文件数据使能
	ReadData: STRING(255) ;//读取的数据
	ReadErrorID: RTS_IEC_RESULT;  //文件读取错误码
	RelReadSize: __XWORD := 0;    //实际读取数据大小，单位字节
//ACT_SysFileWrite 变量	
	xFileWrite: BOOL := FALSE;   //写入文件数据使能
	SentData: STRING := 'This is the first line.SoftVersion:V1.1.$r'; //写入文件内容（$r为回车字符）
	WriteErrorID: RTS_IEC_RESULT;  //文件写入错误码
	RelSentSize: __XWORD := 0;   //实际写入文件数据大小，单位字节
//ACT_SysFileSetPos 变量	
	xFileSetPos: BOOL := FALSE;   //设定文件指针到给定位置
	Offset: __XWORD := 0 ;  //文件指针偏移量
	FileSetPosErrorID: RTS_IEC_RESULT;  //设定文件指针到给定位置错误码	
//ACT_SysFileGetPos 变量
	xFileGetPos: BOOL := FALSE;   //获取文件指针的实际位置
	FileGetPosErrorID: RTS_IEC_RESULT;  //获取文件指针的实际位置错误码
	pulPOS: __XWORD := 1;   //文件指针的实际位置
//ACT_SysFileRename 变量
	xFileRename: BOOL := FALSE;  //重命名文件使能
	OldFileName: STRING := '/usr/src/CODESYSControl/UsrData/test1_copy.txt';    //旧文件路径及文件名
	NewFileName: STRING :='/usr/src/CODESYSControl/UsrData/test2.txt';    //新文件路径及文件名
	FileRenameErrorID: RTS_IEC_RESULT;   //文件重命名错误码
//ACT_SysFileEOF 变量		
	xFileEOF: BOOL := FALSE;  //判断文件内容是否全部读取使能
	FileEOFErrorID: RTS_IEC_RESULT; //ERR_OK表示文件内容已全部读取
//主程序变量表
	iFileState : INT :=0;	  //文件操作步数
	TON_0,TON_1,TON_2:TON; //100ms延时定时器0
	restart: BOOL; //再次启动使能

(*-------------------------------第二部分：记录信息变量---------------------------------------------*)
	sRecordState,sRecordCmd,sRecordError,sRecordSwitch,sRecordXrayState:STRING;		//5组记录的变量
	sRecordTime,sRecordDate,sRecordDateTXT:STRING	;//保存的时间，日期，和文件名
	fbRise			:ARRAY[1..4,1..60] OF R_TRIG;	//触发保存
	fbRiseCmd:R_TRIG;//上位机命令触发保存
	sState,sXrayState:STRING;				//记录日志里显示的内容
	sSwitch1:ARRAY[1..60] OF STRING;	//开关字符串
	sCmd1,sError :ARRAY[1..30] OF STRING;					//命令记录临时字符串
	LS_ReadDintDT_1:LS_SysLib.LS_ReadDintDT;					//获取 PLC 系统时间，将 PLC 系统时间信息存储到内部属性变量中
	bCmd,bError,bState,bSwitch,bXrayState:ARRAY[1..60] OF BOOL;//触发写文件操作
	i,j:INT;//循环变量
	bForceJump:BOOL;//强制跳出，后续不需要了，改为关机时退出
	
(*--------------------------------------第三部分：SD卡相关操作------------------------------------------*)
	LS_CopyToSDCard1:LS_CopyToSDCard;
	SDname:STRING;
	bExe,bDelete,bWrite:BOOL;
	TOF1:TOF;
END_VAR
VAR // added by the converter: edge detectors and wires of the graphical bodies
    _rt1, _rt2, _rt3, _rt4, _rt5, _rt6, _rt7, _rt8 : R_TRIG;
END_VAR


(*readme*)
(*日志记录程序*)
ACT_SysFileOpen();	ACT_SysFileClose();		ACT_SysFileWrite();	ACT_SysFileSetPos();	ACT_SysFileGetPos();
ACT_SysFileRead();	ACT_SysFileEOF();		ACT_SysFileCopy();	ACT_SysFileDelete();	ACT_SysFileRename();

//TOF1(IN:= Entity_IO.bKeySwitch, PT:= T#1S, Q=> bForceJump);//赋值保存

(*1.公共部分，获取系统时间，并转化成字符串形式*)//读取字符串那个功能块有问题，差了8个小时
	LS_ReadDintDT_1(xEnable:= TRUE);
	sRecordTime:=CONCAT(UINT_TO_STRING(LS_ReadDintDT_1.uiYear),'-');
	sRecordTime:=CONCAT(sRecordTime,UINT_TO_STRING(LS_ReadDintDT_1.uiMonth));
	sRecordTime:=CONCAT(sRecordTime,'-');
	sRecordTime:=CONCAT(sRecordTime,UINT_TO_STRING(LS_ReadDintDT_1.uiDay));
	sRecordTime:=CONCAT(sRecordTime,'/');
	sRecordTime:=CONCAT(sRecordTime,UINT_TO_STRING(LS_ReadDintDT_1.uiHour));
	sRecordTime:=CONCAT(sRecordTime,':');
	sRecordTime:=CONCAT(sRecordTime,UINT_TO_STRING(LS_ReadDintDT_1.uiMinute));
	sRecordTime:=CONCAT(sRecordTime,':');
	sRecordTime:=CONCAT(sRecordTime,UINT_TO_STRING(LS_ReadDintDT_1.uiSecond));
	
	sRecordDate:=CONCAT(UINT_TO_STRING(LS_ReadDintDT_1.uiYear),'-');
	sRecordDate:=CONCAT(sRecordDate,UINT_TO_STRING(lS_ReadDintDT_1.uiMonth));
	sRecordDate:=CONCAT(sRecordDate,'-');
	sRecordDate:=CONCAT(sRecordDate,UINT_TO_STRING(LS_ReadDintDT_1.uiDay));
	
	ACT_RecordState();
	ACT_RecordCmd();
	ACT_RecordSwitch();
	ACT_XrayState();
	ACT_RecordError();
	
	
	IF GVL_State.iPLC_State=340 THEN
		bForceJump:=TRUE;
	ELSE
		bForceJump:=FALSE;
	END_IF
	
(*2.文件创建或打开*)
	CASE iFileState OF 
	0:	//复位变量
	  TON_0(IN:= FALSE);TON_1(IN:= FALSE); TON_2(IN:= FALSE);
	  IF GVL_State.iPLC_State>=10 THEN
		iFileState:=10;    
	  END_IF
	  
	10: //打开UsrData目录下文件或者创建文件 “Log.txt”
		PathName :='/usr/src/CODESYSControl/UsrData/Log.txt';  
		xFileOpen := TRUE;
		IF hFile <> RTS_INVALID_HANDLE	THEN    					//文件是否打开判断
			iFileState:=20;
			xFileOpen := FALSE;
		ELSIF  hFile = RTS_INVALID_HANDLE AND OpenErrorID <> 0 THEN 
			iFileState:=100;
			xFileOpen := FALSE;
			RETURN;
		END_IF
		  
	20://在LOG.txt文件内写入数据
		xFileWrite:= TRUE;
		IF RelSentSize <> 0 THEN      	//文件内容是否写入判断
			xFileWrite:= FALSE;
			RelSentSize:=0;       		//复位发送数据大小
			iFileState:=21;
		ELSIF RelSentSize = 0 AND WriteErrorID <>0 THEN 
			iFileState:=100;
			xFileWrite:= FALSE;
			RETURN;
		 END_IF
		 
	21://整机状态记录
		IF bForceJump=FALSE THEN	
			FOR i:=1 TO 15 DO			
				IF bState[i] = TRUE THEN
					iFileState:=20;
					bState[i]:= FALSE;
					SentData := sRecordState;    
					EXIT;
				ELSE
					iFileState:=22;
				END_IF
			END_FOR			
		ELSE
			iFileState:=30;
		END_IF
		
	22://开关量输入记录
		IF bForceJump=FALSE THEN
			FOR i:=1 TO 40 DO			
				IF bSwitch[i] = TRUE THEN
					iFileState:=20;
					bSwitch[i]:= FALSE;
					SentData := sSwitch1[i];   
					EXIT;
				ELSE
					iFileState:=23;		
				END_IF;
			END_FOR
		ELSE
			iFileState:=30;
		END_IF
		
	23://射线源状态记录
		IF bForceJump=FALSE THEN
			FOR i:=1 TO 40 DO			
				IF bXrayState[i] = TRUE THEN
					iFileState:=20;
					bXrayState[i]:= FALSE;
					SentData := sRecordXrayState;   
					EXIT;
				ELSE
					iFileState:=24;		
				END_IF;
			END_FOR
		ELSE
			iFileState:=30;
		END_IF
		
	24://上位机命令记录
		IF bForceJump=FALSE THEN
			FOR i:=1 TO 30 DO 				
				IF bCmd[i] = TRUE THEN
					iFileState:=20;
					bCmd[i]:= FALSE;
					SentData := sCmd1[i];    //写入的数据内容($r为回车字符)
					EXIT;
				ELSE
					iFileState:=25;
				END_IF
			END_FOR			
		ELSE
			iFileState:=30;
		END_IF
		
	25://故障记录
		IF bForceJump=FALSE THEN
			FOR i:=1 TO 5 DO 				
				IF bError[i] = TRUE THEN
					iFileState:=20;
					bError[i]:= FALSE;
					SentData := sError[i];    //写入的数据内容($r为回车字符)
					EXIT;
				ELSE
					iFileState:=21;
				END_IF
			END_FOR			
		ELSE
			iFileState:=30;
		END_IF

	 30: //关闭文件延时判断
	 	//bForceJump:=FALSE;
		bExe:=FALSE;bDelete:=FALSE;
		xFileClose:=TRUE;
		TON_0(IN:= xFileClose, PT:= T#100MS, Q=> , ET=> );  //关闭文件延时判断
		  IF TON_0.Q THEN
			  IF FileCloseErrorID = 0 THEN 
				 xFileClose:=FALSE;   
				 iFileState:=40;
				 hFile := RTS_INVALID_HANDLE;     //必须把文件句柄初始化
			  ELSE  
				xFileClose:=FALSE;
				iFileState:=100;
				RETURN;
			  END_IF 
		  END_IF
			 
	40://写到SD中的文件
		bExe:=TRUE;
		sRecordDateTXT:=CONCAT(sRecordDate,'.txt');
		LS_CopyToSDCard1(
							xExecute:= bExe, 
							strSourceFileName:= 'Log.txt', 
							strDestFileName:= sRecordDateTXT, 
							xDone=> , 
							xError=> , 
							diErrorID=> , 
							dwCopyedSizeBytes=> );
		IF 	LS_CopyToSDCard1.xDone THEN
			iFileState:=50;
			bExe:=FALSE;
		END_IF;			
								
	50://删除文件
		bDelete:=TRUE;
		DelFileName :='/usr/src/CODESYSControl/UsrData/Log.txt';
		xFileDelete:=bDelete;
		  TON_2(IN:= xFileDelete, PT:= T#100MS, Q=> , ET=> );  //删除文件延时判断
		  IF TON_2.Q THEN
			  IF FileDeleteErrorID = 0 THEN 
				 iFileState:=44;
				 xFileDelete :=FALSE; 
			   ELSE  xFileDelete:=FALSE;
					 iFileState:=100;
					 RETURN; 
			  END_IF  
		  END_IF  
   	100:
		;//错误状态

	END_CASE
(*3.文件写入*)

(*4.拷贝文件到SD卡中*)

(*5.关闭文件*)

(*5.删除PLC中的数据记录*)

(*6.关机结束*)

//将 iFileState置为1，开始执行
(*CASE iFileState OF 
	0:
	  ;
	1: //打开UsrData目录下文件或者创建文件 “ test1.txt ”
	  PathName :='/usr/src/CODESYSControl/UsrData/test1.txt';  
      xFileOpen := TRUE;
	  IF hFile <> RTS_INVALID_HANDLE	THEN    //文件是否打开判断
		 iFileState:=2;
		 xFileOpen := FALSE;
	    ELSIF  hFile = RTS_INVALID_HANDLE AND OpenErrorID <> 0 THEN 
			   iFileState:=10;
			   xFileOpen := FALSE;
			   RETURN;
	  END_IF
	  
    2://在test1.txt文件内写入数据
	  SentData := 'This is the first line.$r';    //写入的数据内容($r为回车字符)
	  xFileWrite:= TRUE;
	  IF RelSentSize <> 0 THEN      //文件内容是否写入判断
		 xFileWrite:= FALSE;
         RelSentSize:=0;       //复位发送数据大小
		 iFileState:=3;
		ELSIF RelSentSize = 0 AND WriteErrorID <>0 THEN 
			  iFileState:=10;
			  xFileWrite:= FALSE;
			  RETURN;
	  END_IF
	  ;
	3://设置test1.txt文件指针实际位置
	  Offset:=0;
	  xFileSetPos:= TRUE;
	  xFileGetPos:= TRUE;
	  IF pulPOS=0 AND FileSetPosErrorID = 0 AND FileGetPosErrorID = 0 THEN
		 iFileState:=4;
	     xFileSetPos:= FALSE;
	     xFileGetPos:= FALSE;
	     pulPOS :=1;
      ELSIF  FileSetPosErrorID <> 0 OR FileGetPosErrorID <> 0 THEN 
			 iFileState:=10;
		     xFileSetPos:= FALSE;
	         xFileGetPos:= FALSE;
	         RETURN;
	  END_IF 
	  ;
	4://读取test1.txt文件全部数据内容
	  xFileRead:= TRUE;
	  xFileEOF:= TRUE;
	  IF RelReadSize <> 0 AND FileEOFErrorID= 0 THEN
		 xFileRead:= FALSE;
		 xFileEOF:= FALSE;
		 RelReadSize:=0;
		 iFileState:=5;
	  ELSIF  ReadErrorID <> 0 OR FileEOFErrorID <> 0 THEN 
		     iFileState:=10;
		     xFileRead:= FALSE;
	         xFileEOF:= FALSE;
			 RETURN;
	  END_IF
	  ;
	5://关闭指定文件
	  xFileClose:=TRUE;
	  TON_0(IN:= xFileClose, PT:= T#100MS, Q=> , ET=> );  //关闭文件延时判断
	  IF TON_0.Q THEN
		  IF FileCloseErrorID = 0 THEN 
			 xFileClose:=FALSE;   
             iFileState:=6;
			 hFile := RTS_INVALID_HANDLE;     //必须把文件句柄初始化
          ELSE  xFileClose:=FALSE;
                iFileState:=10;
			    RETURN;
		  END_IF 
	  END_IF
	  ;
	6://复制指定文件
	  CoDestFileName:='/usr/src/CODESYSControl/UsrData/test1_copy.txt';
	  CoSourceFileName :='/usr/src/CODESYSControl/UsrData/test1.txt';
	  xFileCopy:=TRUE;
	  IF CoSize <> 0 AND FileCopyErrorID = 0 THEN
		 xFileCopy:=FALSE;
         CoSize :=0;
         iFileState:=7;
      ELSIF CoSize = 0 AND FileCopyErrorID <> 0 THEN 
			xFileCopy:=FALSE; 
            iFileState:=10;
		    RETURN;
	  END_IF
	  ;
    7://重命名指定文件
	  OldFileName := '/usr/src/CODESYSControl/UsrData/test1_copy.txt';
	  NewFileName := '/usr/src/CODESYSControl/UsrData/test2.txt';   //（若文件名已存在，则报错误码18）
	  xFileRename :=TRUE;        
	  TON_1(IN:= xFileRename, PT:= T#100MS, Q=> , ET=> );  //重命名文件延时判断
	  IF TON_1.Q THEN
		  IF FileRenameErrorID = 0 THEN 
			 iFileState:=8;
             xFileRename :=FALSE;
          ELSE  xFileRename:=FALSE;
                iFileState:=10;
				RETURN;
		  END_IF   
	  END_IF
	  ;
    8://删除指定文件
	  DelFileName :='/usr/src/CODESYSControl/UsrData/test1.txt';
	  xFileDelete:=TRUE;
      TON_2(IN:= xFileDelete, PT:= T#100MS, Q=> , ET=> );  //删除文件延时判断
      IF TON_2.Q THEN
		  IF FileDeleteErrorID = 0 THEN 
			 iFileState:=9;
             xFileDelete :=FALSE; 
		   ELSE  xFileDelete:=FALSE;
                 iFileState:=10;
				 RETURN; 
		  END_IF  
	  END_IF   
	  ;
    9:
      TON_0(IN:= xFileClose, PT:= T#100MS, Q=> , ET=> );    //复位定时器
	  TON_1(IN:= xFileRename, PT:= T#100MS, Q=> , ET=> ); 
	  TON_2(IN:= xFileDelete, PT:= T#100MS, Q=> , ET=> );
      iFileState:=11;  
	  ;
   10:
             //错误状态
	  ; 
   11:
             //完成状态
	  ; 
	  
//执行完一次iFileState循环后，控制器UsrData文件夹内有test2.txt文件，需要删除之后才能再次循环，否则重命名时因文件名已存在会报错	  
IF restart THEN
   DelFileName :='/usr/src/CODESYSControl/UsrData/test2.txt';
   xFileDelete:=TRUE;
   TON_2(IN:= xFileDelete, PT:= T#100MS, Q=> , ET=> );  //删除文件延时判断
      IF TON_2.Q THEN
		  IF FileDeleteErrorID = 0 THEN 
             xFileDelete :=FALSE;
             TON_2(IN:= xFileDelete, PT:= T#10MS, Q=> , ET=> );  //复位定时器
			 restart:=FALSE;
			 iFileState:=1;
			ELSE  xFileDelete:=FALSE;
                  iFileState:=10;
				  RETURN; 
		  END_IF  
	  END_IF 
END_IF         
END_CASE
*)

ACTION ACT_RecordState:

(*记录操作状态变化*)
	sRecordState:=CONCAT(sRecordTime,sState);
	sRecordState:=CONCAT(sRecordState,'.$r');	
		CASE GVL_State.iPLC_State OF 
			10:
				sState:=' _Init';
			20:
				sState:=' _SelfCheck';
			30:
				sState:=' _Homing';
			40:
				sState:=' _Idle';
			110:
				sState:=' _StaticDR';
			120:
				sState:=' _DynamicsDR';
			210:
				sState:=' _StandardCT';
			220:
				sState:=' _StaticCT';
			230:
				sState:=' _HighCT';
			240:
				sState:=' _QuickCT';
			310:
				sState:=' _Error';
			320:
				sState:=' _Debug';
			330:
				sState:=' _Emergency';
			340:
				sState:=' _ShutDown';
		END_CASE
		
		fbRise[1,1](CLK:=GVL_State.iPLC_State=10, Q=> );
		IF fbRise[1,1].Q THEN bState[1]:=TRUE;END_IF
		
		fbRise[1,2](CLK:=GVL_State.iPLC_State=20, Q=> );
		IF fbRise[1,2].Q THEN bState[2]:=TRUE;END_IF
		
		fbRise[1,3](CLK:=GVL_State.iPLC_State=30, Q=> );
		IF fbRise[1,3].Q THEN bState[3]:=TRUE;END_IF
		
		fbRise[1,4](CLK:=GVL_State.iPLC_State=40, Q=> );
		IF fbRise[1,4].Q THEN bState[4]:=TRUE;END_IF
		
		fbRise[1,5](CLK:=GVL_State.iPLC_State=110, Q=> );
		IF fbRise[1,5].Q THEN bState[5]:=TRUE;END_IF
		
		fbRise[1,6](CLK:=GVL_State.iPLC_State=120, Q=> );
		IF fbRise[1,6].Q THEN bState[6]:=TRUE;END_IF
		
		fbRise[1,7](CLK:=GVL_State.iPLC_State=210, Q=> );
		IF fbRise[1,7].Q THEN bState[7]:=TRUE;END_IF
		
		fbRise[1,8](CLK:=GVL_State.iPLC_State=220, Q=> );
		IF fbRise[1,8].Q THEN bState[8]:=TRUE;END_IF
		
		fbRise[1,9](CLK:=GVL_State.iPLC_State=230, Q=> );
		IF fbRise[1,9].Q THEN bState[9]:=TRUE;END_IF
		
		fbRise[1,10](CLK:=GVL_State.iPLC_State=240, Q=> );
		IF fbRise[1,10].Q THEN bState[10]:=TRUE;END_IF
		
		fbRise[1,11](CLK:=GVL_State.iPLC_State=310, Q=> );
		IF fbRise[1,11].Q THEN bState[11]:=TRUE;END_IF
		
		fbRise[1,12](CLK:=GVL_State.iPLC_State=320, Q=> );
		IF fbRise[1,12].Q THEN bState[12]:=TRUE;END_IF
		
		fbRise[1,13](CLK:=GVL_State.iPLC_State=330, Q=> );
		IF fbRise[1,13].Q THEN bState[13]:=TRUE;END_IF
		
		fbRise[1,14](CLK:=GVL_State.iPLC_State=340, Q=> );
		IF fbRise[1,14].Q THEN bState[14]:=TRUE;END_IF
END_ACTION

ACTION ACT_RecordError:


(*1.旋转电机报错*)
	fbRise[3,1](CLK:=Axis_XZ.XZ_AxisState.ErrorID<>0, Q=> );
	IF fbRise[3,1].Q THEN bError[1]:=TRUE;
		sError[1]:=CONCAT(sRecordTime,' Axis_XZ.Error:');
		sError[1]:=CONCAT(sError[1],UDINT_TO_STRING(WorkStation_TCP.XZ_Error));
		sError[1]:=CONCAT(sError[1],'.$r');
	END_IF

(*2.前进电机报错*)
	fbRise[3,2](CLK:=Axis_QJ.QJ_AxisState.ErrorID<>0, Q=> );
	IF fbRise[3,2].Q THEN bError[2]:=TRUE;
		sError[2]:=CONCAT(sRecordTime,' Axis_QJ.Error:');
		sError[2]:=CONCAT(sError[2],UDINT_TO_STRING(WorkStation_TCP.QJ_Error));
		sError[2]:=CONCAT(sError[2],'.$r');
	END_IF;

(*3.射线源报错*)
	fbRise[3,3](CLK:=DT_Xray.iAlarmNum<>0, Q=> );
	IF fbRise[3,3].Q THEN bError[3]:=TRUE;
		sError[3]:=CONCAT(sRecordTime,' Xray.Error:');
		sError[3]:=CONCAT(sError[3],UINT_TO_STRING(DT_Xray.iAlarmNum));
		sError[3]:=CONCAT(sError[3],'.$r');
	END_IF;
END_ACTION

ACTION ACT_RecordCmd:



(*记录命令变化*)
	sRecordCmd:=CONCAT(sRecordTime,'.$r');
	
	fbRiseCmd(CLK:=(WorkStation_TCP.PLC_RECV_TEMP.m_nSocketType = 1),Q=> );
	IF fbRiseCmd.Q THEN
		FOR j:=1 TO 27 BY 1 DO 
			bCmd[j]:=TRUE;
		END_FOR
	END_IF;
	
	(*1*)
	sCmd1[1]:=CONCAT(sRecordTime,':$r');
	(*2*)
	sCmd1[2]:=CONCAT('	m_nExpId:',UDINT_TO_STRING(WorkStation_TCP.PLC_RECV_TEMP.m_nExpId));
	sCmd1[2]:=CONCAT(sCmd1[2],'.$r');
	(*3*)
	sCmd1[3]:=CONCAT('	m_nAngleStart:',REAL_TO_STRING(WorkStation_TCP.PLC_RECV_TEMP.m_nAngleStart));
	sCmd1[3]:=CONCAT(sCmd1[3],'.$r');
	(*4*)
	sCmd1[4]:=CONCAT('	m_nAngleEnd:',REAL_TO_STRING(WorkStation_TCP.PLC_RECV_TEMP.m_nAngleEnd));
	sCmd1[4]:=CONCAT(sCmd1[4],'.$r');
	(*5*)
	sCmd1[5]:=CONCAT('	m_nRotateBegin:',REAL_TO_STRING(WorkStation_TCP.PLC_RECV_TEMP.m_nRotateBegin));
	sCmd1[5]:=CONCAT(sCmd1[5],'.$r');
	(*6*)
	sCmd1[6]:=CONCAT('	m_nRotateEnd:',REAL_TO_STRING(WorkStation_TCP.PLC_RECV_TEMP.m_nRotateEnd));
	sCmd1[6]:=CONCAT(sCmd1[6],'.$r');
	(*7*)
	sCmd1[7]:=CONCAT('	m_nKv:',UDINT_TO_STRING(WorkStation_TCP.PLC_RECV_TEMP.m_nKv));
	sCmd1[7]:=CONCAT(sCmd1[7],'.$r');
	(*8*)
	sCmd1[8]:=CONCAT('	m_nMA:',REAL_TO_STRING(WorkStation_TCP.PLC_RECV_TEMP.m_nMA));
	sCmd1[8]:=CONCAT(sCmd1[8],'.$r');
	(*9*)
	sCmd1[9]:=CONCAT('	m_nMS:',REAL_TO_STRING(WorkStation_TCP.PLC_RECV_TEMP.m_nMS));
	sCmd1[9]:=CONCAT(sCmd1[9],'.$r');
	(*10*)
	sCmd1[10]:=CONCAT('	m_nFocus:',UDINT_TO_STRING(WorkStation_TCP.PLC_RECV_TEMP.m_nFocus));
	sCmd1[10]:=CONCAT(sCmd1[10],'.$r');
	(*11*)
	sCmd1[11]:=CONCAT('	m_nAcquireFrame:',UDINT_TO_STRING(WorkStation_TCP.PLC_RECV_TEMP.m_nAcquireFrame));
	sCmd1[11]:=CONCAT(sCmd1[11],'.$r');
	(*12*)
	sCmd1[12]:=CONCAT('	m_nFramePerCirCle:',UDINT_TO_STRING(WorkStation_TCP.PLC_RECV_TEMP.m_nFramePerCirCle));
	sCmd1[12]:=CONCAT(sCmd1[12],'.$r');
	(*13*)
	sCmd1[13]:=CONCAT('	m_nMoveToward:',UDINT_TO_STRING(WorkStation_TCP.PLC_RECV_TEMP.m_nMoveToward));
	sCmd1[13]:=CONCAT(sCmd1[13],'.$r');
	(*14*)
	sCmd1[14]:=CONCAT('	m_nScanUseType:',UDINT_TO_STRING(WorkStation_TCP.PLC_RECV_TEMP.m_nServenLamp));
	sCmd1[14]:=CONCAT(sCmd1[14],'.$r');
	(*15*)
	sCmd1[15]:=CONCAT('	m_nMoveStep:',REAL_TO_STRING(WorkStation_TCP.PLC_RECV_TEMP.m_nMoveStep));
	sCmd1[15]:=CONCAT(sCmd1[15],'.$r');
	(*16*)
	sCmd1[16]:=CONCAT('	m_nPitchValue:',REAL_TO_STRING(WorkStation_TCP.PLC_RECV_TEMP.m_nPitchValue));
	sCmd1[16]:=CONCAT(sCmd1[16],'.$r');
	(*17*)
	sCmd1[17]:=CONCAT('	m_nCircleCount:',UDINT_TO_STRING(WorkStation_TCP.PLC_RECV_TEMP.m_nCircleCount));
	sCmd1[17]:=CONCAT(sCmd1[17],'.$r');
	(*18*)
	sCmd1[18]:=CONCAT('	m_nControlState:',UDINT_TO_STRING(WorkStation_TCP.PLC_RECV_TEMP.m_nControlState));
	sCmd1[18]:=CONCAT(sCmd1[18],'.$r');
	(*19*)
	sCmd1[19]:=CONCAT('	m_fScanTop:',REAL_TO_STRING(WorkStation_TCP.PLC_RECV_TEMP.m_fScanTop));
	sCmd1[19]:=CONCAT(sCmd1[19],'.$r');
	(*20*)
	sCmd1[20]:=CONCAT('	m_fScanBottom:',REAL_TO_STRING(WorkStation_TCP.PLC_RECV_TEMP.m_fScanBottom));
	sCmd1[20]:=CONCAT(sCmd1[20],'.$r');
	(*21*)
	sCmd1[21]:=CONCAT('	m_fSecondPerCicle:',REAL_TO_STRING(WorkStation_TCP.PLC_RECV_TEMP.m_fSecondPerCicle));
	sCmd1[21]:=CONCAT(sCmd1[21],'.$r');
	(*22*)
	sCmd1[22]:=CONCAT('	m_nSamplingRate:',UDINT_TO_STRING(WorkStation_TCP.PLC_RECV_TEMP.m_nSamplingRate));
	sCmd1[22]:=CONCAT(sCmd1[22],'.$r');
	(*23*)
	sCmd1[23]:=CONCAT('	m_nPrepareState:',UDINT_TO_STRING(WorkStation_TCP.PLC_RECV_TEMP.m_nPrepareState));
	sCmd1[23]:=CONCAT(sCmd1[23],'.$r');
	(*24*)
	sCmd1[24]:=CONCAT('	m_nScanMoveType:',UDINT_TO_STRING(WorkStation_TCP.PLC_RECV_TEMP.m_nScanMoveType));
	sCmd1[24]:=CONCAT(sCmd1[24],'.$r');
	(*25*)
	sCmd1[25]:=CONCAT('	m_nCircleIndex:',UDINT_TO_STRING(WorkStation_TCP.PLC_RECV_TEMP.m_nCircleIndex));
	sCmd1[25]:=CONCAT(sCmd1[25],'.$r');
	(*26*)
	sCmd1[26]:=CONCAT('	m_nPLCMaCoeff:',REAL_TO_STRING(WorkStation_TCP.PLC_RECV_TEMP.m_nPLCMaCoeff));
	sCmd1[26]:=CONCAT(sCmd1[26],'.$r');
	(*27*)
	sCmd1[27]:=CONCAT('	m_nLastMsg:',UDINT_TO_STRING(WorkStation_TCP.PLC_RECV_TEMP.m_nLastMsg));
	sCmd1[27]:=CONCAT(sCmd1[27],'.$r');
	(*28*)
	sCmd1[28]:=CONCAT('	m_nDelayTime:',UDINT_TO_STRING(WorkStation_TCP.PLC_RECV_TEMP.m_nDelayTime));
	sCmd1[28]:=CONCAT(sCmd1[28],'.$r');
END_ACTION

ACTION ACT_XrayState:

(*记录操作状态变化*)
	sRecordXrayState:=CONCAT(sRecordTime,sXrayState);
	sRecordXrayState:=CONCAT(sRecordXrayState,'.$r');	
		CASE GVL_State.iXray_State OF 
			10:
				sXrayState:=' Xray_OpenSeria';
			20:
				sXrayState:=' Xray_Init';
			30:
				sXrayState:=' Xray_DefaultPara';
			40:
				sXrayState:=' Xray_QueryState';
			50:
				sXrayState:=' Xray_ExposurePara';
			60:
				sXrayState:=' Xray_Exposure';
			70:
				sXrayState:=' Xray_FluoroPara';
			80:
				sXrayState:=' Xray_FluoroExPosure';
			90:
				sXrayState:=' Xray_DrPara';
			100:
				sXrayState:=' Xray_DrExposure';
			44:
				sXrayState:=' Xray_Error';
			
		END_CASE
		
		fbRise[4,1](CLK:=GVL_State.iXray_State=10, Q=> );
		IF fbRise[4,1].Q THEN bXrayState[1]:=TRUE;END_IF
		
		fbRise[4,2](CLK:=GVL_State.iXray_State=20, Q=> );
		IF fbRise[4,2].Q THEN bXrayState[2]:=TRUE;END_IF
		
		fbRise[4,3](CLK:=GVL_State.iXray_State=30, Q=> );
		IF fbRise[4,3].Q THEN bXrayState[3]:=TRUE;END_IF
		
		fbRise[4,4](CLK:=GVL_State.iXray_State=40, Q=> );
		IF fbRise[4,4].Q THEN bXrayState[4]:=TRUE;END_IF
		
		fbRise[4,5](CLK:=GVL_State.iXray_State=50, Q=> );
		IF fbRise[4,5].Q THEN bXrayState[5]:=TRUE;END_IF
		
		fbRise[4,6](CLK:=GVL_State.iXray_State=60, Q=> );
		IF fbRise[4,6].Q THEN bXrayState[6]:=TRUE;END_IF
		
		fbRise[4,7](CLK:=GVL_State.iXray_State=70, Q=> );
		IF fbRise[4,7].Q THEN bXrayState[7]:=TRUE;END_IF
		
		fbRise[4,8](CLK:=GVL_State.iXray_State=80, Q=> );
		IF fbRise[4,8].Q THEN bXrayState[8]:=TRUE;END_IF
		
		fbRise[4,9](CLK:=GVL_State.iXray_State=90, Q=> );
		IF fbRise[4,9].Q THEN bXrayState[9]:=TRUE;END_IF
		
		fbRise[4,10](CLK:=GVL_State.iXray_State=100, Q=> );
		IF fbRise[4,10].Q THEN bXrayState[10]:=TRUE;END_IF
		
		fbRise[4,11](CLK:=GVL_State.iXray_State=44, Q=> );
		IF fbRise[4,11].Q THEN bXrayState[11]:=TRUE;END_IF
END_ACTION

ACTION ACT_SysFileOpen:
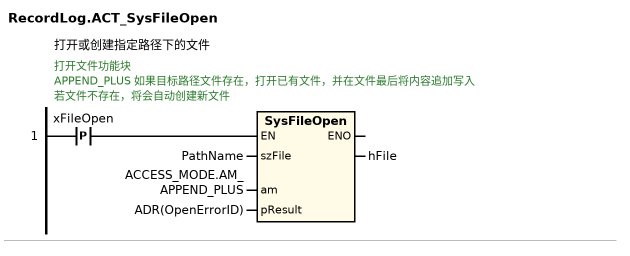
// NETWORK 1: 打开或创建指定路径下的文件
// 打开文件功能块
// APPEND_PLUS 如果目标路径文件存在，打开已有文件，并在文件最后将内容追加写入
//             若文件不存在，将会自动创建新文件
_rt1(CLK := xFileOpen);
IF _rt1.Q THEN
    hFile := SysFileOpen(szFile := PathName, am := ACCESS_MODE.AM_APPEND_PLUS, pResult := ADR(OpenErrorID));
END_IF
END_ACTION

ACTION ACT_SysFileRename:
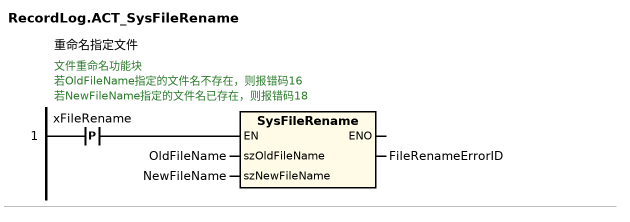
// NETWORK 1: 重命名指定文件
// 文件重命名功能块
// 若OldFileName指定的文件名不存在，则报错码16
// 若NewFileName指定的文件名已存在，则报错码18
_rt2(CLK := xFileRename);
IF _rt2.Q THEN
    FileRenameErrorID := SysFileRename(szOldFileName := OldFileName, szNewFileName := NewFileName);
END_IF
END_ACTION

ACTION ACT_SysFileRead:
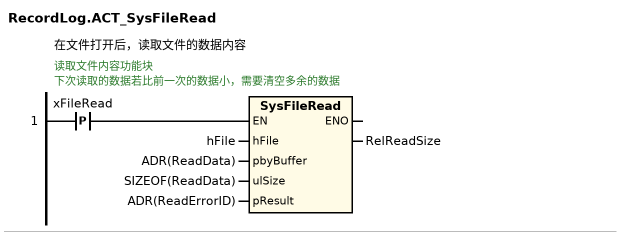
// NETWORK 1: 在文件打开后，读取文件的数据内容
// 读取文件内容功能块
// 下次读取的数据若比前一次的数据小，需要清空多余的数据
_rt3(CLK := xFileRead);
IF _rt3.Q THEN
    RelReadSize := SysFileRead(hFile := hFile, pbyBuffer := ADR(ReadData), ulSize := SIZEOF(ReadData), pResult := ADR(ReadErrorID));
END_IF
END_ACTION

ACTION ACT_SysFileDelete:
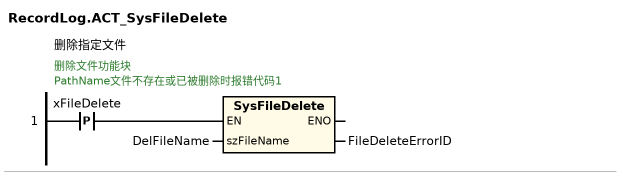
// NETWORK 1: 删除指定文件
// 删除文件功能块
// PathName文件不存在或已被删除时报错代码1
_rt4(CLK := xFileDelete);
IF _rt4.Q THEN FileDeleteErrorID := SysFileDelete(szFileName := DelFileName); END_IF
END_ACTION

ACTION ACT_SysFileSetPos:
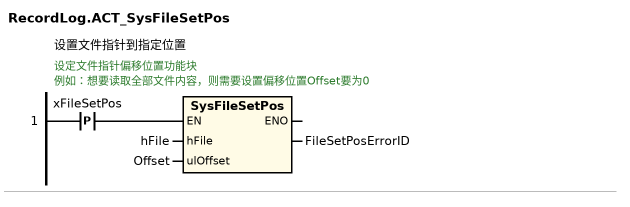
// NETWORK 1: 设置文件指针到指定位置
// 设定文件指针偏移位置功能块
// 例如：想要读取全部文件内容，则需要设置偏移位置Offset要为0
_rt5(CLK := xFileSetPos);
IF _rt5.Q THEN FileSetPosErrorID := SysFileSetPos(hFile := hFile, ulOffset := Offset); END_IF
END_ACTION

ACTION ACT_SysFileWrite:
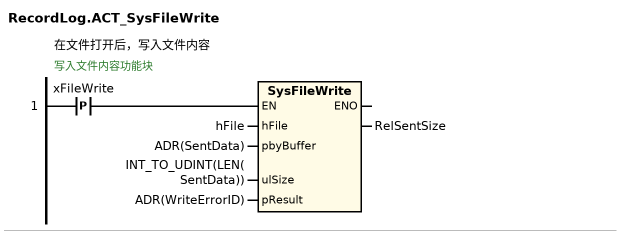
// NETWORK 1: 在文件打开后，写入文件内容
// 写入文件内容功能块
_rt6(CLK := xFileWrite);
IF _rt6.Q THEN
    RelSentSize := SysFileWrite(hFile := hFile, pbyBuffer := ADR(SentData), ulSize := INT_TO_UDINT(LEN(SentData)), pResult := ADR(WriteErrorID));
END_IF
END_ACTION

ACTION ACT_SysFileClose:
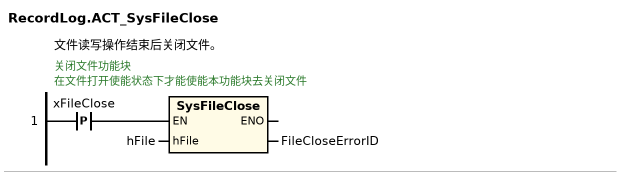
// NETWORK 1: 文件读写操作结束后关闭文件。
// 关闭文件功能块
// 在文件打开使能状态下才能使能本功能块去关闭文件
_rt7(CLK := xFileClose);
IF _rt7.Q THEN FileCloseErrorID := SysFileClose(hFile := hFile); END_IF
END_ACTION

ACTION ACT_SysFileEOF:
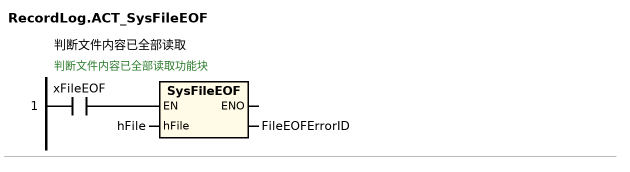
// NETWORK 1: 判断文件内容已全部读取
// 判断文件内容已全部读取功能块
IF xFileEOF THEN FileEOFErrorID := SysFileEOF(hFile := hFile); END_IF
END_ACTION

ACTION ACT_SysFileGetPos:
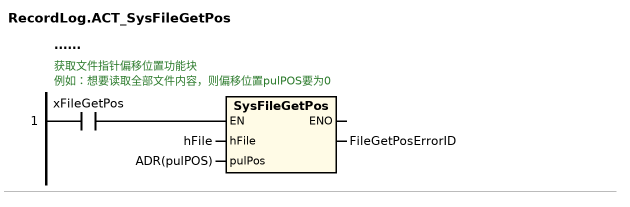
// NETWORK 1: ......
// 获取文件指针偏移位置功能块
// 例如：想要读取全部文件内容，则偏移位置pulPOS要为0
IF xFileGetPos THEN FileGetPosErrorID := SysFileGetPos(hFile := hFile, pulPos := ADR(pulPOS)); END_IF
END_ACTION

ACTION ACT_SysFileCopy:
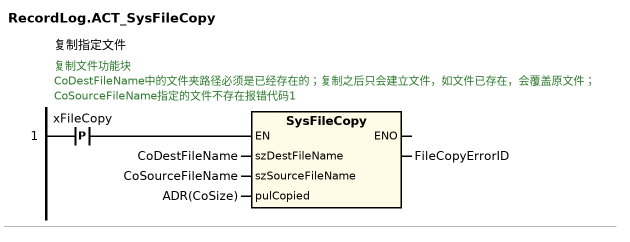
// NETWORK 1: 复制指定文件
// 复制文件功能块
// CoDestFileName中的文件夹路径必须是已经存在的；复制之后只会建立文件，如文件已存在，会覆盖原文件；
// CoSourceFileName指定的文件不存在报错代码1
_rt8(CLK := xFileCopy);
IF _rt8.Q THEN
    FileCopyErrorID := SysFileCopy(szDestFileName := CoDestFileName, szSourceFileName := CoSourceFileName, pulCopied := ADR(CoSize));
END_IF
END_ACTION

ACTION ACT_RecordSwitch:


(*开关操作日志*)
	(*-------------------------------------第一部分，左右PANNEL-------------------------------------*)
		fbRise[2,1](CLK:=Entity_IO.LeftPannel_BedUp, Q=> );
		IF fbRise[2,1].Q THEN bSwitch[1]:=TRUE;
			sSwitch1[1]:=CONCAT(sRecordTime,'.LeftPannel_BedUp');
			sSwitch1[1]:=CONCAT(sSwitch1[1],'.$r');
		END_IF
		
		fbRise[2,2](CLK:=Entity_IO.LeftPannel_BedDown, Q=> );
		IF fbRise[2,2].Q THEN bSwitch[2]:=TRUE;
			sSwitch1[2]:=CONCAT(sRecordTime,'.LeftPannel_BedDown');
			sSwitch1[2]:=CONCAT(sSwitch1[2],'.$r');
		END_IF
		
		fbRise[2,3](CLK:=Entity_IO.LeftPannel_BedFore, Q=> );
		IF fbRise[2,3].Q THEN bSwitch[3]:=TRUE;
			sSwitch1[3]:=CONCAT(sRecordTime,'.LeftPannel_BedFore');
			sSwitch1[3]:=CONCAT(sSwitch1[3],'.$r');
		END_IF
		
		fbRise[2,4](CLK:=Entity_IO.LeftPannel_BedBack, Q=> );
		IF fbRise[2,4].Q THEN bSwitch[4]:=TRUE;
			sSwitch1[4]:=CONCAT(sRecordTime,'.LeftPannel_BedBack');
			sSwitch1[4]:=CONCAT(sSwitch1[4],'.$r');
		END_IF
		
		fbRise[2,5](CLK:=Entity_IO.LeftPannel_LaserButton, Q=> );
		IF fbRise[2,5].Q THEN bSwitch[5]:=TRUE;
			sSwitch1[5]:=CONCAT(sRecordTime,'.LeftPannel_LaserButton');
			sSwitch1[5]:=CONCAT(sSwitch1[5],'.$r');
		END_IF
		
		fbRise[2,6](CLK:=Entity_IO.LeftPannel_DistanceMove, Q=> );
		IF fbRise[2,6].Q THEN bSwitch[6]:=TRUE;
			sSwitch1[6]:=CONCAT(sRecordTime,'.LeftPannel_MoveZero');
			sSwitch1[6]:=CONCAT(sSwitch1[6],'.$r');
		END_IF
		
		fbRise[2,7](CLK:=Entity_IO.LeftPannel_RecordPos, Q=> );
		IF fbRise[2,7].Q THEN bSwitch[7]:=TRUE;
			sSwitch1[7]:=CONCAT(sRecordTime,'.LeftPannel_RecordPos');
			sSwitch1[7]:=CONCAT(sSwitch1[7],'.$r');
		END_IF
		
		fbRise[2,8](CLK:=Entity_IO.LeftPannel_MoveRecordPos, Q=> );
		IF fbRise[2,8].Q THEN bSwitch[8]:=TRUE;
			sSwitch1[8]:=CONCAT(sRecordTime,'.LeftPannel_MoveRecordPos');
			sSwitch1[8]:=CONCAT(sSwitch1[8],'.$r');
		END_IF
		
		fbRise[2,9](CLK:=Entity_IO.RightPannel_BedUp, Q=> );
		IF fbRise[2,9].Q THEN bSwitch[9]:=TRUE;
			sSwitch1[9]:=CONCAT(sRecordTime,'.RightPannel_BedUp');
			sSwitch1[9]:=CONCAT(sSwitch1[9],'.$r');
		END_IF
		
		fbRise[2,10](CLK:=Entity_IO.RightPannel_BedDown, Q=> );
		IF fbRise[2,10].Q THEN bSwitch[10]:=TRUE;
			sSwitch1[10]:=CONCAT(sRecordTime,'.RightPannel_BedDown');
			sSwitch1[10]:=CONCAT(sSwitch1[10],'.$r');
		END_IF
		
		fbRise[2,11](CLK:=Entity_IO.RightPannel_BedFore, Q=> );
		IF fbRise[2,11].Q THEN bSwitch[11]:=TRUE;
			sSwitch1[11]:=CONCAT(sRecordTime,'.RightPannel_BedFore');
			sSwitch1[11]:=CONCAT(sSwitch1[11],'.$r');
		END_IF
		
		fbRise[2,12](CLK:=Entity_IO.RightPannel_BedBack, Q=> );
		IF fbRise[2,12].Q THEN bSwitch[12]:=TRUE;
			sSwitch1[12]:=CONCAT(sRecordTime,'.RightPannel_BedBack');
			sSwitch1[12]:=CONCAT(sSwitch1[12],'.$r');
		END_IF
		
		fbRise[2,13](CLK:=Entity_IO.RightPannel_LaserButton, Q=> );
		IF fbRise[2,13].Q THEN bSwitch[13]:=TRUE;
			sSwitch1[13]:=CONCAT(sRecordTime,'.RightPannel_LaserButton');
			sSwitch1[13]:=CONCAT(sSwitch1[13],'.$r');
		END_IF
		
		fbRise[2,14](CLK:=Entity_IO.RightPannel_DistanceMove, Q=> );
		IF fbRise[2,14].Q THEN bSwitch[14]:=TRUE;
			sSwitch1[14]:=CONCAT(sRecordTime,'.RightPannel_MoveZero');
			sSwitch1[14]:=CONCAT(sSwitch1[14],'.$r');
		END_IF
		
		fbRise[2,15](CLK:=Entity_IO.RightPannel_RecordPos, Q=> );
		IF fbRise[2,15].Q THEN bSwitch[15]:=TRUE;
			sSwitch1[15]:=CONCAT(sRecordTime,'.RightPannel_RecordPos');
			sSwitch1[15]:=CONCAT(sSwitch1[15],'.$r');
		END_IF
		
		fbRise[2,16](CLK:=Entity_IO.RightPannel_MoveRecordPos, Q=> );
		IF fbRise[2,16].Q THEN bSwitch[16]:=TRUE;
			sSwitch1[16]:=CONCAT(sRecordTime,'.RightPannel_MoveRecordPos');
			sSwitch1[16]:=CONCAT(sSwitch1[16],'.$r');
		END_IF
		
	(*-------------------------------------第二部分，CTBOX-------------------------------------*)	
		fbRise[2,17](CLK:=CTBOX_RS232.CTBOX_KEY_Manual, Q=> );
		IF fbRise[2,17].Q THEN bSwitch[17]:=TRUE;
			sSwitch1[17]:=CONCAT(sRecordTime,'.CTBOX_KEY_Manual');
			sSwitch1[17]:=CONCAT(sSwitch1[17],'.$r');
		END_IF
		
		fbRise[2,18](CLK:=CTBOX_RS232.CTBOX_KEY_Auto, Q=> );
		IF fbRise[2,18].Q THEN bSwitch[18]:=TRUE;
			sSwitch1[18]:=CONCAT(sRecordTime,'.CTBOX_KEY_Auto');
			sSwitch1[18]:=CONCAT(sSwitch1[18],'.$r');
		END_IF
		
		fbRise[2,19](CLK:=CTBOX_RS232.CTBOX_KEY_Stop, Q=> );
		IF fbRise[2,19].Q THEN bSwitch[19]:=TRUE;
			sSwitch1[19]:=CONCAT(sRecordTime,'.CTBOX_KEY_Stop');
			sSwitch1[19]:=CONCAT(sSwitch1[19],'.$r');
		END_IF
		
		fbRise[2,20](CLK:=CTBOX_RS232.CTBOX_KEY_MoveDistance, Q=> );
		IF fbRise[2,20].Q THEN bSwitch[20]:=TRUE;
			sSwitch1[20]:=CONCAT(sRecordTime,'.CTBOX_KEY_MoveDistance');
			sSwitch1[20]:=CONCAT(sSwitch1[20],'.$r');
		END_IF
		
		fbRise[2,21](CLK:=CTBOX_RS232.CTBOX_KEY_BedFore, Q=> );
		IF fbRise[2,21].Q THEN bSwitch[21]:=TRUE;
			sSwitch1[21]:=CONCAT(sRecordTime,'.CTBOX_KEY_BedFore');
			sSwitch1[21]:=CONCAT(sSwitch1[21],'.$r');
		END_IF
		
		fbRise[2,22](CLK:=CTBOX_RS232.CTBOX_KEY_BedUp, Q=> );
		IF fbRise[2,22].Q THEN bSwitch[22]:=TRUE;
			sSwitch1[22]:=CONCAT(sRecordTime,'.CTBOX_KEY_BedUp');
			sSwitch1[22]:=CONCAT(sSwitch1[22],'.$r');
		END_IF
		
		fbRise[2,23](CLK:=CTBOX_RS232.CTBOX_KEY_BedBack, Q=> );
		IF fbRise[2,23].Q THEN bSwitch[23]:=TRUE;
			sSwitch1[23]:=CONCAT(sRecordTime,'.CTBOX_KEY_BedBack');
			sSwitch1[23]:=CONCAT(sSwitch1[23],'.$r');
		END_IF
		
		fbRise[2,24](CLK:=CTBOX_RS232.CTBOX_KEY_BedDown, Q=> );
		IF fbRise[2,24].Q THEN bSwitch[24]:=TRUE;
			sSwitch1[24]:=CONCAT(sRecordTime,'.CTBOX_KEY_BedDown');
			sSwitch1[24]:=CONCAT(sSwitch1[24],'.$r');
		END_IF
		
		(*-------------------------------------第三部分，其他IO-------------------------------------*)	
(*		fbRise[2,25](CLK:=Entity_IO.bUpMotorMin, Q=> );
		IF fbRise[2,25].Q THEN bSwitch[25]:=TRUE;
			sSwitch1[25]:=CONCAT(sRecordTime,'.bUpMotorMin');
			sSwitch1[25]:=CONCAT(sSwitch1[25],'.$r');
		END_IF
		
		fbRise[2,26](CLK:=Entity_IO.bUpMotorSTO, Q=> );
		IF fbRise[2,26].Q THEN bSwitch[26]:=TRUE;
			sSwitch1[26]:=CONCAT(sRecordTime,'.bUpMotorSTO');
			sSwitch1[26]:=CONCAT(sSwitch1[26],'.$r');
		END_IF
*)		
		fbRise[2,27](CLK:=Entity_IO.bXrayOneInput, Q=> );
		IF fbRise[2,27].Q THEN bSwitch[27]:=TRUE;
			sSwitch1[27]:=CONCAT(sRecordTime,'.bXrayOneInput');
			sSwitch1[27]:=CONCAT(sSwitch1[27],'.$r');
		END_IF
		
		fbRise[2,28](CLK:=Entity_IO.bXrayTwoInput, Q=> );
		IF fbRise[2,28].Q THEN bSwitch[28]:=TRUE;
			sSwitch1[28]:=CONCAT(sRecordTime,'.bXrayTwoInput');
			sSwitch1[28]:=CONCAT(sSwitch1[28],'.$r');
		END_IF
		
		fbRise[2,29](CLK:=Entity_IO.bXrayFluInput, Q=> );
		IF fbRise[2,29].Q THEN bSwitch[29]:=TRUE;
			sSwitch1[29]:=CONCAT(sRecordTime,'.bXrayFluInput');
			sSwitch1[29]:=CONCAT(sSwitch1[29],'.$r');
		END_IF
		
		fbRise[2,30](CLK:=Entity_IO.bXayExpoInput, Q=> );
		IF fbRise[2,30].Q THEN bSwitch[30]:=TRUE;
			sSwitch1[30]:=CONCAT(sRecordTime,'.bXayExpoInput');
			sSwitch1[30]:=CONCAT(sSwitch1[30],'.$r');
		END_IF
		
		fbRise[2,31](CLK:=Entity_IO.bKeySwitch, Q=> );
		IF fbRise[2,31].Q THEN bSwitch[31]:=TRUE;
			sSwitch1[31]:=CONCAT(sRecordTime,'.bKeySwitch');
			sSwitch1[31]:=CONCAT(sSwitch1[31],'.$r');
		END_IF
		
		(*新增TriggerOut输出记录功能1229*)
		IF GVL_State.iPLC_State=110 OR GVL_State.iPLC_State=220 THEN //静态DR和静态CT，记录TRIGGER输出
			fbRise[2,32](CLK:=Entity_IO.bTriggerOut, Q=> );
			IF fbRise[2,32].Q THEN bSwitch[32]:=TRUE;
				sSwitch1[32]:=CONCAT(sRecordTime,'.Entity_IO.bSync_In');
				sSwitch1[32]:=CONCAT(sSwitch1[32],'.$r');
			END_IF
		END_IF;
	
		fbRise[2,33](CLK:=Entity_IO.bEmergencyStop, Q=> );
		IF fbRise[2,33].Q THEN bSwitch[33]:=TRUE;
			sSwitch1[33]:=CONCAT(sRecordTime,'.bEmergencyStop');
			sSwitch1[33]:=CONCAT(sSwitch1[33],'.$r');
		END_IF
		
		(*新增探测器sync_out输出记录功能0106*)
		IF GVL_State.iPLC_State=110 OR GVL_State.iPLC_State=220 THEN //静态DR和静态CT，记录TRIGGER输出
			fbRise[2,34](CLK:=Entity_IO.bSync_out, Q=> );
			IF fbRise[2,34].Q THEN bSwitch[34]:=TRUE;
				sSwitch1[34]:=CONCAT(sRecordTime,'.Entity_IO.bSync_Out');
				sSwitch1[34]:=CONCAT(sSwitch1[34],'.$r');
			END_IF
		END_IF;
(*		
		fbRise[2,34](CLK:=Entity_IO.bXzMotorSTO, Q=> );
		IF fbRise[2,34].Q THEN bSwitch[34]:=TRUE;
			sSwitch1[34]:=CONCAT(sRecordTime,'.bXzMotorSTO');
			sSwitch1[34]:=CONCAT(sSwitch1[34],'.$r');
		END_IF
*)		
		fbRise[2,35](CLK:=Entity_IO.bForeMotorMin, Q=> );
		IF fbRise[2,35].Q THEN bSwitch[35]:=TRUE;
			sSwitch1[35]:=CONCAT(sRecordTime,'.bForeMotorMin');
			sSwitch1[35]:=CONCAT(sSwitch1[35],'.$r');
		END_IF
		
		fbRise[2,36](CLK:=Entity_IO.bForeMotorMax, Q=> );
		IF fbRise[2,36].Q THEN bSwitch[36]:=TRUE;
			sSwitch1[36]:=CONCAT(sRecordTime,'.bForeMotorMax');
			sSwitch1[36]:=CONCAT(sSwitch1[36],'.$r');
		END_IF
		
		fbRise[2,37](CLK:=Entity_IO.bRotateMotorMin, Q=> );
		IF fbRise[2,37].Q THEN bSwitch[37]:=TRUE;
			sSwitch1[37]:=CONCAT(sRecordTime,'.bRotateMotorMin');
			sSwitch1[37]:=CONCAT(sSwitch1[37],'.$r');
		END_IF
		
		fbRise[2,38](CLK:=Entity_IO.bRotateMotorMax, Q=> );
		IF fbRise[2,38].Q THEN bSwitch[38]:=TRUE;
			sSwitch1[38]:=CONCAT(sRecordTime,'.bRotateMotorMax');
			sSwitch1[38]:=CONCAT(sSwitch1[38],'.$r');
		END_IF
		
		fbRise[2,39](CLK:=Entity_IO.bCalibrate, Q=> );
		IF fbRise[2,39].Q THEN bSwitch[39]:=TRUE;
			sSwitch1[39]:=CONCAT(sRecordTime,'.bCalibrate');
			sSwitch1[39]:=CONCAT(sSwitch1[39],'.$r');
		END_IF
END_ACTION

END_PROGRAM

// Device/Application/Communication/Calibration
PROGRAM Calibration
VAR
	count:BYTE;
	i:INT;
	abyReadData:ARRAY[0..119] OF BYTE;
	iLength:INT;
	j: INT;
	Num:INT;
END_VAR

(*readme*)
(*标定功能块*)
(*	IF WorkStation_TCP.TCP_Read_1.xDone THEN
		FOR i:=0 TO 20 BY 1 DO 
			IF abyReadData[i]=16#0A THEN
				iLength:=i;
				EXIT;
			END_IF
		END_FOR
	ELSE
		;
	END_IF
	
	FOR j:=0 TO 20 BY 1 DO
		IF abyReadData[i]=16#30 THEN
			Num:=0;
		ELSIF abyReadData[i]=16#31 THEN
			Num:=1;
		ELSIF abyReadData[i]=16#32 THEN
			Num:=2;
		ELSIF abyReadData[i]=16#33 THEN
			Num:=3;
		ELSIF abyReadData[i]=16#34 THEN
			Num:=4;
		ELSIF abyReadData[i]=16#35 THEN
			Num:=5;
		ELSIF abyReadData[i]=16#36 THEN
			Num:=6;
		ELSIF abyReadData[i]=16#37 THEN
			Num:=7;
		ELSIF abyReadData[i]=16#38 THEN
			Num:=5;
		ELSIF abyReadData[i]=16#39 THEN
			Num:=6;
		ELSIF abyReadData[i]=16#37 THEN
			Num:=7;
		
		END_IF
		
	END_FOR
	
	
	CASE i OF 
	0:
	;
	1:
	;
	2:
	;
	3:
	;
	4:
	
	END_CASE
	
	
	
	
	
	
	
	
	
	IF abyReadData[0]=*)

END_PROGRAM

// Device/Application/BasicFBs/MoveFilter
FUNCTION_BLOCK MoveFilter
VAR_INPUT
	Input:INT;
	N:INT;
END_VAR
VAR_OUTPUT
	Output:INT;
END_VAR
VAR
	Sum:INT;
	CO: INT;
END_VAR


Input:=0;

CO:=Input*N;
Sum:=Sum-Input+CO;
Output:=Sum/N;

END_FUNCTION_BLOCK

// Device/Application/BasicFBs/RC
FUNCTION_BLOCK RC
VAR_EXTERNAL

END_VAR

VAR_INPUT
	Input:UINT;
END_VAR
VAR_OUTPUT
	Output:UINT;
END_VAR
VAR
	prev:UINT;
END_VAR

(*======================== READ_ME ==============================*)
(*功能块：“低通滤波”                                           	 *)
(*=========================== END ===============================*)
prev:=UDINT_TO_UINT(6*UINT_TO_UDINT(Input)/10+4*UINT_TO_UDINT(prev)/10);
Output:=prev;

END_FUNCTION_BLOCK

// Device/Application/BasicFBs/Curve_Cs
FUNCTION_BLOCK Curve_Cs
VAR_EXTERNAL

END_VAR

VAR_INPUT
	X_Array	:ARRAY [ 0..9 ] OF INT;
	Y_Array	:ARRAY [ 0..9 ] OF INT;
	length	:INT;	
	Value_X	:INT;
END_VAR

VAR_OUTPUT
	Value_Y	:INT;
	Error:bool;
END_VAR

VAR
	BOOTING:BOOL:=0;
	POS_OR_NEG:bool;
	COUNT_NUM:INT:=0;
	COUNT_OLD:INT;
	TEMP_Length:INT;
END_VAR

(*============================ READ_ME ================================*)
(*功能块：“分段线性化曲线”                                           *)
(*根据给出的传感器分度表，进行分段线性计算，得出当前阻值对应的工程量   *)
(*注意，横坐标“X_Array”应从数组元素[0]开始按照从小到大的顺序写入值   *)
(*注意，length为写入数组元素的个数                                     *)
(*============================== END ==================================*)
	IF BOOTING=0 THEN
		IF ((X_Array[1]-X_Array[0])>0 AND (Y_Array[1]-Y_Array[0])>0) or ( (X_Array[1]-X_Array[0])<0 AND (Y_Array[1]-Y_Array[0])<0 ) THEN
			POS_OR_NEG:=1;
		ELSIF ((X_Array[1]-X_Array[0])>0 AND (Y_Array[1]-Y_Array[0])<0) or ( (X_Array[1]-X_Array[0])<0 AND (Y_Array[1]-Y_Array[0])>0 ) THEN
			POS_OR_NEG:=0;
		END_IF;		
		BOOTING:=1;
	END_IF;

	IF length<=1 or length>10 THEN
		TEMP_Length:=9;
	ELSE
		TEMP_Length:=length-1;
	END_IF;
	IF POS_OR_NEG=0 THEN
		IF COUNT_NUM<(TEMP_Length-1) THEN
			COUNT_NUM:=COUNT_NUM+1;
		ELSE
			COUNT_NUM:=0;
		END_IF;		
	ELSE
		IF COUNT_NUM>0 THEN
			COUNT_NUM:=COUNT_NUM-1;
		ELSE
			COUNT_NUM:=TEMP_Length-1;
		END_IF;		
	END_IF;
	COUNT_OLD:=COUNT_NUM+1;
	
	IF X_Array[COUNT_NUM]<X_Array[COUNT_OLD] and Error=0 THEN
		IF (Value_X>X_Array[COUNT_NUM]) AND (Value_X<=X_Array[COUNT_OLD]) THEN
			Value_Y:=Y_Array[COUNT_NUM]+dint_to_int(int_to_dint(Y_Array[COUNT_OLD]-Y_Array[COUNT_NUM])*int_to_dint(Value_X-X_Array[COUNT_NUM])/int_to_dint(X_Array[COUNT_OLD]-X_Array[COUNT_NUM]));
			IF POS_OR_NEG=1 THEN
				COUNT_NUM:=TEMP_Length-1;
			ELSE
				COUNT_NUM:=0;
			END_IF;				
		ELSIF Value_X<=X_Array[0] THEN
			Value_Y:=Y_Array[0];
		ELSIF Value_X>X_Array[TEMP_Length] THEN
			Value_Y:=Y_Array[TEMP_Length];		
		END_IF;	
	ELSE
		Error:=1;
		Value_Y:=0;
	END_IF;

END_FUNCTION_BLOCK

// Device/Application/Refer/WriteLog
PROGRAM WriteLog
VAR
//ACT_SysFileOpen 变量
    xFileOpen: BOOL := FALSE;  //打开文件使能
	PathName: STRING := '/usr/src/CODESYSControl/UsrData/test1.txt';  //文件路径及文件名
	OpenErrorID: RTS_IEC_RESULT;   //文件打开错误码
	hFile: RTS_IEC_HANDLE := RTS_INVALID_HANDLE;  //文件句柄
//ACT_SysFileClose 变量	
	xFileClose: BOOL := FALSE;   //关闭文件使能
	FileCloseErrorID: RTS_IEC_RESULT;  //文件关闭错误码
//ACT_SysFileCopy 变量	
	xFileCopy: BOOL := FALSE; //复制文件使能
	CoDestFileName: STRING :='/usr/src/CODESYSControl/UsrData/test1_copy.txt' ; //目标文件路径及文件名
	CoSourceFileName: STRING := '/usr/src/CODESYSControl/UsrData/test1.txt';  //源文件路径及文件名
	CoSize: __XWORD := 0;  //实际复制文件大小，单位字节
	FileCopyErrorID: RTS_IEC_RESULT :=0;   //文件复制错误码
//ACT_SysFileDelete 变量
	xFileDelete: BOOL := FALSE;  //删除文件使能
	DelFileName: STRING :='/usr/src/CODESYSControl/UsrData/test1.txt';  //删除的文件路径及文件名
	FileDeleteErrorID: RTS_IEC_RESULT;  //文件删除错误码
//ACT_SysFileRead 变量	
	xFileRead: BOOL := FALSE;   //读取文件数据使能
	ReadData: STRING(128) ;//读取的数据
	ReadErrorID: RTS_IEC_RESULT;  //文件读取错误码
	RelReadSize: __XWORD := 0;    //实际读取数据大小，单位字节
//ACT_SysFileWrite 变量	
	xFileWrite: BOOL := FALSE;   //写入文件数据使能
	SentData: STRING(128) := 'This is the first line.$r'; //写入文件内容（$r为回车字符）
	WriteErrorID: RTS_IEC_RESULT;  //文件写入错误码
	RelSentSize: __XWORD := 0;   //实际写入文件数据大小，单位字节
//ACT_SysFileSetPos 变量	
	xFileSetPos: BOOL := FALSE;   //设定文件指针到给定位置
	Offset: __XWORD := 0 ;  //文件指针偏移量
	FileSetPosErrorID: RTS_IEC_RESULT;  //设定文件指针到给定位置错误码	
//ACT_SysFileGetPos 变量
	xFileGetPos: BOOL := FALSE;   //获取文件指针的实际位置
	FileGetPosErrorID: RTS_IEC_RESULT;  //获取文件指针的实际位置错误码
	pulPOS: __XWORD := 1;   //文件指针的实际位置
//ACT_SysFileRename 变量
	xFileRename: BOOL := FALSE;  //重命名文件使能
	OldFileName: STRING := '/usr/src/CODESYSControl/UsrData/test1_copy.txt';    //旧文件路径及文件名
	NewFileName: STRING :='/usr/src/CODESYSControl/UsrData/test2.txt';    //新文件路径及文件名
	FileRenameErrorID: RTS_IEC_RESULT;   //文件重命名错误码
//ACT_SysFileEOF 变量		
	xFileEOF: BOOL := FALSE;  //判断文件内容是否全部读取使能
	FileEOFErrorID: RTS_IEC_RESULT; //ERR_OK表示文件内容已全部读取
//主程序变量表
	iFileState : INT :=0;	  //文件操作步数
	TON_0:TON; //100ms延时定时器0
	TON_1:TON; //100ms延时定时器1
	TON_2:TON; //100ms延时定时器2
	restart: BOOL; //再次启动使能
	
END_VAR
VAR // added by the converter: edge detectors and wires of the graphical bodies
    _rt1, _rt2, _rt3, _rt4, _rt5, _rt6, _rt7, _rt8 : R_TRIG;
END_VAR

//本例程用于演示控制器目录下的文件管理功能

ACT_SysFileOpen();
ACT_SysFileClose();
ACT_SysFileWrite();
ACT_SysFileSetPos();
ACT_SysFileGetPos();
ACT_SysFileRead();
ACT_SysFileEOF();
ACT_SysFileCopy();
ACT_SysFileDelete();
ACT_SysFileRename();

//将 iFileState置为1，开始执行
CASE iFileState OF 
	0:
	  ;
	1: //打开UsrData目录下文件或者创建文件 “ test1.txt ”
	  PathName :='/usr/src/CODESYSControl/UsrData/test1.txt';  
      xFileOpen := TRUE;
	  IF hFile <> RTS_INVALID_HANDLE	THEN    //文件是否打开判断
		 iFileState:=2;
		 xFileOpen := FALSE;
	    ELSIF  hFile = RTS_INVALID_HANDLE AND OpenErrorID <> 0 THEN 
			   iFileState:=10;
			   xFileOpen := FALSE;
			   RETURN;
	  END_IF
	  
